No03: NOP   0;
NoXX: NOP   0;
NETWORK
TITLE =ASW_6030: Active step germinating
//      U     "MAL1S019Par".Par.FlagProcess.ProcessActive;
//      SPBN  tuen;
//
//// copy stepnr
//      L     "MAL1S019Par".Par.ParIntMachine.ActualStep;
//      T     "MAL1S019Par".Par.ParIntProcess.ActualStep;
//// set step conditions
//
//// Case where process is starting during loading
//      U     "MAL1S019Par".Par.FlagProcess.ProcessActive;
//      UN    "MAL1S019Par".Par.FlagFunction_1.StepLoading; // Step loading
//      SPBN  e003;
//// lifting devices must be in highest position
//      L       WinCoS_BIW01_09PLC1BIW01_02.Ma.Par.ParPositionTopRightUnits;
////Malting Plant OAO Belsolod Ivanonvo Weissrussland
//      L     50; // 50mm offset
//      +I    ;
//      T     "MAL1S019Par".Par.MachineValue.SOLLWERT_HUBZUG1_HOEHE;
//      L       WinCoS_BIW01_09PLC1BIW01_02.Ma.Par.ParPositionTopLeftUnits;
////Malting Plant OAO Belsolod Ivanonvo Weissrussland
//      L     50; // 50mm offset
//      +I    ;
//      T     "MAL1S019Par".Par.MachineValue.SOLLWERT_HUBZUG2_HOEHE;
//      L     5;
//      T     WinCoS_BIW01_09PLC1BIW01_02.Ma.Par.ParTolPosition;
//e003: NOP   0;
//
//// reset turning cmds
//
//// save turning cmds from prev.step
//      L     "MAL1S019Par".Par.ParIntMachine.ActualStep;
//      L     "MAL1S019Par".Par.ParIntProcess.PrevStep1stTurn;
//      <>I   ;
//      SPB   sav1;
//      U     "MAL1S019Par".Par.FlagProcess2.Turning1WithSpraying;
//      =     "MAL1S019Par".Par.Switches1.StaOn08; // Turning1WithSpraying
//      U     "MAL1S019Par".Par.FlagProcess2.Turning1WithDosing;
//      =     "MAL1S019Par".Par.Switches1.StaOn09; // Turning1WithDosing
//sav1: NOP   0;
//      L     "MAL1S019Par".Par.ParIntMachine.ActualStep;
//      L     "MAL1S019Par".Par.ParIntProcess.PrevStep2ndTurn;
//      <>I   ;
//      SPB   sav2;
//      U     "MAL1S019Par".Par.FlagProcess2.Turning2WithSpraying;
//      =     "MAL1S019Par".Par.Switches1.StaOn10; // Turning2WithSpraying
//      U     "MAL1S019Par".Par.FlagProcess2.Turning2WithDosing;
//      =     "MAL1S019Par".Par.Switches1.StaOn11; // Turning2WithDosing
//sav2: NOP   0;
//
//      SET   ;
//      R     "MAL1S019Par".Par.FlagProcess2.Turning1WithoutSpraying;
//      R     "MAL1S019Par".Par.FlagProcess2.Turning1WithSpraying;
//      R     "MAL1S019Par".Par.FlagProcess2.Turning1WithDosing;
//      R     "MAL1S019Par".Par.FlagProcess2.Turning2WithoutSpraying;
//      R     "MAL1S019Par".Par.FlagProcess2.Turning2WithSpraying;
//      R     "MAL1S019Par".Par.FlagProcess2.Turning2WithDosing;
//
//// Delta Temp to switch to next step
//      L     "MAL1S019Par".StepAct.DeltaTempSwitchpointStep;
//      L     L#0;
//      >D   ;
//      =     "MAL1S019Par".Par.FlagProcess1.DeltaTempNextStep;
//// Max Temp to switch to next step
//      L     "MAL1S019Par".StepAct.MaxTempAboveFloorStep;
//      L     L#0;
//      >D   ;
//      =     "MAL1S019Par".Par.FlagProcess1.MaxTempNextStep;
//
//// position waste air see sub 6050
//
//// basic speed fan see sub 6040
//
//// air humifidication
//      L     1;
//      L     "MAL1S019Par".StepAct.AirMoisten;   // On/Off
//      ==I;  // air humifidication on
//      U     WinCoS_BIW01_09PLC1BIW01_02.Ma.StStartedFwd; //Malting Plant OAO
//Belsolod Ivanonvo Weissrussland
//      =     "MAL1S019Par".Par.FlagProcess.AirHumidificationValve1; // air
//humifidication valve 1 on
//      U(    ; // air humifidication on
//      L     "MAL1S019Par".Par.ParIntMachine.TargetSpeedGermFan; // germinating
//fan is running
//      L     40; // fanspeed > 40%
//      >I    ; // muss noch in Istwert getauscht werden JV
//      )     ; // fanspeed > 40%
//      =     "MAL1S019Par".Par.FlagProcess.AirHumidificationValve2;
//
//// air cooling
//      L     "MAL1S019Par".StepAct.Cooling;
//      L   1;  // Activate Cooling System = 1 (yes)
//      ==I;
//      =     "MAL1S019Par".Par.FlagProcess.Cooling; // request cooling
//
//      U     "MAL1S019Par".Par.FlagProcess.ProcessActive;
//      U     "MAL1S019".PCRead.Step.StReady;
//      UN    "MAL1S019Par".Par.FlagFunction_1.StepLoading;
//      SPBN  e630;
//
//// turning 1
//      UN    "MAL1S019Par".Par.FlagProcess2.StartSecondTurningRound; // Turn
//from PrevStep
//      U(;
//      L     "MAL1S019Par".StepAct.StartTurningRound_1;
//      L     0;
//      >=D;                  // negative, no turning 1
//      );
//      U(    ;
//      O(    ; // Nach Rezept
//      L     "MAL1S019Par".ActTimeStepProcess.StepTimeActHourTotal; // Steptime
//in hours overall
//      L     "MAL1S019Par".StepAct.StartTurningRound_1;
//      ==I   ;
//      UN     WinCoS_BIW01_09PLC1BIW01_02.Ma.StAdjusted; // target position
//turning reached
//      )     ;
//      O(    ; // Selbsthaltung
//      L     "MAL1S019Par".ActTimeStepProcess.StepTimeActHourTotal; // Steptime
//in hours overall
//      L     "MAL1S019Par".StepAct.StartTurningRound_1;
//      <>I   ;
//      U     "MAL1S019Par".Par.FlagProcess2.StartFirstTurningRound;
//      )     ;
//      )     ;
//      S     "MAL1S019Par".Par.FlagProcess2.Turning1WithoutSpraying;
//      S     "MAL1S019Par".Par.FlagFunction_1.TurningStart;
//// turning 1 with spraying
//      U(    ;
//      L     1;
//      L     "MAL1S019Par".StepAct.TurningWithSpraying_1;
//      ==I;    // turning 1 with spraying on
//      U(    ;
//      L     "MAL1S019Par".Par.ParIntMachine.ActualStep;
//      L     "MAL1S019Par".Par.ParIntProcess.PrevStep1stTurn;
//      ==I   ;
//      )     ;
//      )     ;
//      O(    ;
//      L     "MAL1S019Par".Par.ParIntMachine.ActualStep;
//      L     "MAL1S019Par".Par.ParIntProcess.PrevStep1stTurn;
//      <>I   ;
//      U     "MAL1S019Par".Par.Switches1.StaOn08; // Turning1WithSpraying
//      )     ;
//      U     "MAL1S019Par".Par.FlagProcess2.Turning1WithoutSpraying;
//      S     "MAL1S019Par".Par.FlagProcess2.Turning1WithSpraying;
//// turning 1 with spraying and GA3
//      U(    ;
//      L     1;
//      L     "MAL1S019Par".StepAct.TurningWithDosing_1;
//      ==I;    // turning 1 with spraying on
//      U(    ;
//      L     "MAL1S019Par".Par.ParIntMachine.ActualStep;
//      L     "MAL1S019Par".Par.ParIntProcess.PrevStep1stTurn;
//      ==I   ;
//      )     ;
//      )     ;
//      O(    ;
//      L     "MAL1S019Par".Par.ParIntMachine.ActualStep;
//      L     "MAL1S019Par".Par.ParIntProcess.PrevStep1stTurn;
//      <>I   ;
//      U     "MAL1S019Par".Par.Switches1.StaOn09; // Turning1WithDosing
//      )     ;
//      U     "MAL1S019Par".Par.FlagProcess2.Turning1WithoutSpraying;
//      S     "MAL1S019Par".Par.FlagProcess2.Turning1WithSpraying;
//      S     "MAL1S019Par".Par.FlagProcess2.Turning1WithDosing;
//
//      U     "MAL1S019Par".Par.FlagProcess2.Turning1WithoutSpraying;
//      U     "MAL1S019Par".Par.FlagFunction_1.TurningStart;
//      UN     WinCoS_BIW01_09PLC1BIW01_02.Ma.StAdjusted; // target position
//turning reached
//      FP    "MAL1S019Par".Par.FlagProcess2.StartFirstTurningFP;
//      S     "MAL1S019Par".Par.FlagProcess2.StartFirstTurningRound;
//
//      U     WinCoS_BIW01_09PLC1BIW01_02.Ma.StAdjusted; // target position
//turning reached
//      O(    ;
//      L     "MAL1S019Par".ActTimeStepProcess.StepTimeActHourTotal; // Steptime
//in hours overall
//      L     "MAL1S019Par".StepAct.StartTurningRound_1;
//      >I    ;
//      U     WinCoS_BIW01_09PLC1BIW01_02.Ma.StAdjusted; // target position
//turning reached
//      )     ;
//      U     "MAL1S019Par".Par.FlagProcess2.StartFirstTurningRound;
//      R     "MAL1S019Par".Par.FlagProcess2.StartFirstTurningRound;
//
//      U     "MAL1S019Par".Par.FlagProcess2.StartFirstTurningFP;
//      SPB   trn1;
//      L     "MAL1S019Par".Par.ParIntMachine.ActualStep;
//      T     "MAL1S019Par".Par.ParIntProcess.PrevStep1stTurn;
//trn1: NOP   0;
//
//// turning 2
//      UN    "MAL1S019Par".Par.FlagProcess2.StartFirstTurningRound; // Unsinngie
//Rezeptwerte
//      U(;
//      L     1;
//      L     "MAL1S019Par".StepAct.StartTurningRound_2;
//      ==I    ;
//      );
//      U(    ;
//      O(    ; // Nach Rezept
//      L     "MAL1S019Par".ActTimeStepProcess.StepTimeActHourTotal; // Steptime
//in hours overall
//      L     "MAL1S019Par".StepAct.StartTurningRound_2;
//      ==I   ;
//      UN     WinCoS_BIW01_09PLC1BIW01_02.Ma.StAdjusted; // target position
//turning reached
//      )     ;
//      O(    ; // Selbsthaltung
//      L     "MAL1S019Par".ActTimeStepProcess.StepTimeActHourTotal; // Steptime
//in hours overall
//      L     "MAL1S019Par".StepAct.StartTurningRound_2;
//      <>I   ;
//      U     "MAL1S019Par".Par.FlagProcess2.StartSecondTurningRound;
//      )     ;
//      )     ;
//      S     "MAL1S019Par".Par.FlagProcess2.Turning2WithoutSpraying;
//      S     "MAL1S019Par".Par.FlagFunction_1.TurningStart;
//// turning 2 with spraying
//      U(    ;
//      L     1;
//      L     "MAL1S019Par".StepAct.TurningWithSpraying_2;
//      ==I    ;
//      U(    ;
//      L     "MAL1S019Par".Par.ParIntMachine.ActualStep;
//      L     "MAL1S019Par".Par.ParIntProcess.PrevStep2ndTurn;
//      ==I   ;
//      )     ;
//      )     ;
//      O(    ;
//      L     "MAL1S019Par".Par.ParIntMachine.ActualStep;
//      L     "MAL1S019Par".Par.ParIntProcess.PrevStep2ndTurn;
//      <>I   ;
//      U     "MAL1S019Par".Par.Switches1.StaOn10; // Turning2WithSpraying
//      )     ;
//      U     "MAL1S019Par".Par.FlagProcess2.Turning2WithoutSpraying;
//      S     "MAL1S019Par".Par.FlagProcess2.Turning2WithSpraying;
//// turning 2 with spraying and GA3
//      U(    ;
//      L     1;
//      L     "MAL1S019Par".StepAct.TurningWithDosing_2;
//      ==I;    // turning 2 with spraying and GA3 on
//      U(    ;
//      L     "MAL1S019Par".Par.ParIntMachine.ActualStep;
//      L     "MAL1S019Par".Par.ParIntProcess.PrevStep2ndTurn;
//      ==I   ;
//      )     ;
//      )     ;
//      O(    ;
//      L     "MAL1S019Par".Par.ParIntMachine.ActualStep;
//      L     "MAL1S019Par".Par.ParIntProcess.PrevStep2ndTurn;
//      <>I   ;
//      U     "MAL1S019Par".Par.Switches1.StaOn11; // Turning2WithDosing
//      )     ;
//      U     "MAL1S019Par".Par.FlagProcess2.Turning2WithoutSpraying;
//      S     "MAL1S019Par".Par.FlagProcess2.Turning2WithSpraying;
//      S     "MAL1S019Par".Par.FlagProcess2.Turning2WithDosing;
//
//      U     "MAL1S019Par".Par.FlagProcess2.Turning2WithoutSpraying;
//      U     "MAL1S019Par".Par.FlagFunction_1.TurningStart;
//      UN     WinCoS_BIW01_09PLC1BIW01_02.Ma.StAdjusted; // target position
//turning reached
//      FP    "MAL1S019Par".Par.FlagProcess2.StartSecondTurningFP;
//      S     "MAL1S019Par".Par.FlagProcess2.StartSecondTurningRound;
//
//      U     WinCoS_BIW01_09PLC1BIW01_02.Ma.StAdjusted; // target position
//turning reached
//      O(    ;
//      L     "MAL1S019Par".ActTimeStepProcess.StepTimeActHourTotal; // Steptime
//in hours overall
//      L     "MAL1S019Par".StepAct.StartTurningRound_2;
//      >I    ;
//      U     WinCoS_BIW01_09PLC1BIW01_02.Ma.StAdjusted; // target position
//turning reached
//      )     ;
//      U     "MAL1S019Par".Par.FlagProcess2.StartSecondTurningRound;
//      R     "MAL1S019Par".Par.FlagProcess2.StartSecondTurningRound;
//
//      U     "MAL1S019Par".Par.FlagProcess2.StartSecondTurningFP;
//      SPB   trn2;
//      L     "MAL1S019Par".Par.ParIntMachine.ActualStep;
//      T     "MAL1S019Par".Par.ParIntProcess.PrevStep2ndTurn;
//trn2: NOP   0;
////Fix Speed for Turning
//      U     "MAL1S019Par".Par.FlagProcess2.Turning1WithoutSpraying;
//      O     "MAL1S019Par".Par.FlagProcess2.Turning1WithSpraying;
//      O     "MAL1S019Par".Par.FlagProcess2.Turning2WithoutSpraying;
//      O     "MAL1S019Par".Par.FlagProcess2.Turning2WithSpraying;
//      U    M 50.0;
//      SPBN  SpdT;
//      L     15; // 15Hz
//      T     "MAL1S019Par".Par.MachineValue.SollwertFahrantrieb;
//SpdT: NOP   0;
//
//// find turning direction
//      U     "MAL1S019Par".Par.FlagGen.TurningStarted;
//      O(    ;
//      UN    "MAL1S019Par".Par.FlagProcess2.Turning1WithoutSpraying;
//      UN    "MAL1S019Par".Par.FlagProcess2.Turning2WithoutSpraying;
//      )     ;
//      SPB   tuen;
//      L     "MAL1S019Par".Par.ParIntMachine.TargetPosTravDriTurnRigt; // 370° =
//endposition turning right
//      T     WinCoS_BIW01_09PLC1BIW01_02.Ma.InPositionTarget; // target position
//turning reached
//
//      U(    ;
//      L     WinCoS_BIW01_09PLC1BIW01_02.Ma.OutPositionAngle;
//      L     1800;
//      <I    ; // condition turning right (clockwise)
//      )     ;
//      S     "MAL1S019Par".Par.FlagFunction_1.TurningRight;
//      S     "MAL1S019Par".Par.FlagGen.TurningStarted;
//// - Correct effect of ILO Mode
//      L       WinCoS_BIW01_09PLC1BIW01_02.Ma.Par.ParPositionTopLeftUnits;
////Malting Plant OAO Belsolod Ivanonvo Weissrussland
//      T     "MAL1S019Par".Par.MachineValue.SOLLWERT_HUBZUG1_HOEHE;
//      L       WinCoS_BIW01_09PLC1BIW01_02.Ma.Par.ParPositionTopRightUnits;
////Malting Plant OAO Belsolod Ivanonvo Weissrussland
//      T     "MAL1S019Par".Par.MachineValue.SOLLWERT_HUBZUG2_HOEHE;
//      SPB   E603   ;
//      L     "MAL1S019Par".Par.ParIntMachine.TargetPosTravDriTurnLeft; // 0° =
//endposition turning left
//      T     WinCoS_BIW01_09PLC1BIW01_02.Ma.InPositionTarget; // target position
//turning reached
//
//      U(    ;
//      L     WinCoS_BIW01_09PLC1BIW01_02.Ma.OutPositionAngle;
//      L     1800;
//      >=I   ; // condition turning left (counterclockwise)
//      )     ;
//      S     "MAL1S019Par".Par.FlagFunction_1.TurningLeft;
//      S     "MAL1S019Par".Par.FlagGen.TurningStarted;
//// - Correct effect of ILO Mode
//      L       WinCoS_BIW01_09PLC1BIW01_02.Ma.Par.ParPositionTopLeftUnits;
////Malting Plant OAO Belsolod Ivanonvo Weissrussland
//      T     "MAL1S019Par".Par.MachineValue.SOLLWERT_HUBZUG1_HOEHE;
//      L       WinCoS_BIW01_09PLC1BIW01_02.Ma.Par.ParPositionTopRightUnits;
////Malting Plant OAO Belsolod Ivanonvo Weissrussland
//      T     "MAL1S019Par".Par.MachineValue.SOLLWERT_HUBZUG2_HOEHE;
//      SPB   E603   ;
//tuen: NOP   0;
//// - Case of fast speed to protect a 2nd start during same hours as finsihed
//      O(    ; // Nach Rezept
//      L     "MAL1S019Par".ActTimeStepProcess.StepTimeActHourTotal; // Steptime
//in hours overall
//      L     "MAL1S019Par".StepAct.StartTurningRound_1;
//      ==I   ;
//      U     WinCoS_BIW01_09PLC1BIW01_02.Ma.StAdjusted; // target position
//turning reached
//      U     "MAL1S019Par".Par.FlagFunction_1.TurningStart;
//      )     ;
//      O(    ; // Nach Rezept
//      L     "MAL1S019Par".ActTimeStepProcess.StepTimeActHourTotal; // Steptime
//in hours overall
//      L     "MAL1S019Par".StepAct.StartTurningRound_2;
//      ==I   ;
//      U     WinCoS_BIW01_09PLC1BIW01_02.Ma.StAdjusted; // target position
//turning reached
//      U     "MAL1S019Par".Par.FlagFunction_1.TurningStart;
//      )     ;
//      SPB   e603;
//
//// reset turning right (clockwise)
//      U     "MAL1S019Par".Par.FlagFunction_1.TurningRight;
//      U(    ;
//      O      WinCoS_BIW01_09PLC1BIW01_02.Ma.StAdjusted; // target position
//turning reached
//      O(    ;
//      L     WinCoS_BIW01_09PLC1BIW01_02.Ma.OutPositionAngle;
//      L     WinCoS_BIW01_09PLC1BIW01_02.Ma.Par.ParTolPosition;
//      +I    ;
//      L     "MAL1S019Par".Par.ParIntMachine.TargetPosTravDriTurnRigt;
//      >=I   ;
//      )     ;
//      )     ;
//      R     "MAL1S019Par".Par.FlagFunction_1.TurningRight;
//      R     "MAL1S019Par".Par.FlagFunction_1.TurningStart;
//
//// reset turning left (counterclockwise)
//      U     "MAL1S019Par".Par.FlagFunction_1.TurningLeft;
//      U(    ;
//      O     WinCoS_BIW01_09PLC1BIW01_02.Ma.StAdjusted; // target position
//turning reached
//      O(    ;
//      L     WinCoS_BIW01_09PLC1BIW01_02.Ma.OutPositionAngle;
//      L     WinCoS_BIW01_09PLC1BIW01_02.Ma.Par.ParTolPosition;
//      -I    ;
//      L     "MAL1S019Par".Par.ParIntMachine.TargetPosTravDriTurnLeft;
//      <=I   ;
//      )     ;
//      )     ;
//      R     "MAL1S019Par".Par.FlagFunction_1.TurningLeft;
//      R     "MAL1S019Par".Par.FlagFunction_1.TurningStart;
//
//// reset turning flag
//      U     "MAL1S019Par".Par.FlagGen.TurningStarted;
//      UN    "MAL1S019Par".Par.FlagProcess2.Turning1WithoutSpraying;
//      UN    "MAL1S019Par".Par.FlagProcess2.Turning2WithoutSpraying;
//      O(    ;
//      U     "MAL1S019Par".Par.FlagGen.TurningStarted;
//      U     WinCoS_BIW01_09PLC1BIW01_02.Ma.StAdjusted; // target position
//turning reached
//      )     ;
//      ON    "MAL1S019Par".Par.FlagProcess.ProcessActive;
//      R     "MAL1S019Par".Par.FlagGen.TurningStarted;
//      R     "MAL1S019Par".Par.FlagProcess2.Turning1WithoutSpraying;
//      R     "MAL1S019Par".Par.FlagProcess2.Turning2WithoutSpraying;
//      R     "MAL1S019Par".Par.FlagFunction_1.TurningStart;
//e630: NOP   0;
//      UN    "MAL1S019Par".Par.FlagProcess.ProcessActive;
//      R     "MAL1S019Par".Par.FlagProcess2.StartFirstTurningRound;
//      R     "MAL1S019Par".Par.FlagProcess2.StartSecondTurningRound;
//
//e603: NOP   0;
//E603: NOP   0;

      A     "MAL1S019Par".Par.FlagProcess.ProcessActive;
      JCN   tuen;

// copy stepnr
      L     "MAL1S019Par".Par.ParIntMachine.ActualStep;
      T     "MAL1S019Par".Par.ParIntProcess.ActualStep;
// set step conditions

// reset turning cmds

// save turning cmds from prev.step
      L     "MAL1S019Par".Par.ParIntMachine.ActualStep;
      L     "MAL1S019Par".Par.ParIntProcess.PrevStep1stTurn;
      <>I   ;
      JC    sav1;
      A     "MAL1S019Par".Par.FlagProcess2.Turning1WithSpraying;
      =     "MAL1S019Par".Par.Switches1.StaOn08; // Turning1WithSpraying
      A     "MAL1S019Par".Par.FlagProcess2.Turning1WithDosing;
      =     "MAL1S019Par".Par.Switches1.StaOn09; // Turning1WithDosing
sav1: NOP   0;
      L     "MAL1S019Par".Par.ParIntMachine.ActualStep;
      L     "MAL1S019Par".Par.ParIntProcess.PrevStep2ndTurn;
      <>I   ;
      JC    sav2;
      A     "MAL1S019Par".Par.FlagProcess2.Turning2WithSpraying;
      =     "MAL1S019Par".Par.Switches1.StaOn10; // Turning2WithSpraying
      A     "MAL1S019Par".Par.FlagProcess2.Turning2WithDosing;
      =     "MAL1S019Par".Par.Switches1.StaOn11; // Turning2WithDosing
sav2: NOP   0;

      SET   ;
      R     "MAL1S019Par".Par.FlagProcess2.Turning1WithoutSpraying;
      R     "MAL1S019Par".Par.FlagProcess2.Turning1WithSpraying;
      R     "MAL1S019Par".Par.FlagProcess2.Turning1WithDosing;
      R     "MAL1S019Par".Par.FlagProcess2.Turning2WithoutSpraying;
      R     "MAL1S019Par".Par.FlagProcess2.Turning2WithSpraying;
      R     "MAL1S019Par".Par.FlagProcess2.Turning2WithDosing;

// Delta Temp to switch to next step
      L     "MAL1S019Par".StepAct.DeltaTempSwitchpointStep;
      L     L#0;
      >D    ;
      =     "MAL1S019Par".Par.FlagProcess1.DeltaTempNextStep;
// Max Temp to switch to next step
      L     "MAL1S019Par".StepAct.MaxTempAboveFloorStep;
      L     L#0;
      >D    ;
      =     "MAL1S019Par".Par.FlagProcess1.MaxTempNextStep;

// position waste air see sub 6050

// basic speed fan see sub 6040

// air humifidication

// air cooling
      L     "MAL1S019Par".StepAct.Cooling;
      L     1; // Activate Cooling System = 1 (yes)
      ==I   ;
      =     "MAL1S019Par".Par.FlagProcess.Cooling; // request cooling

      A     "MAL1S019Par".Par.FlagProcess.ProcessActive;
      A     "MAL1S019".PCRead.Step.StReady;
      AN    "MAL1S019Par".Par.FlagFunction_1.StepLoading;
      JCN   e630;

// turning 1
      AN    "MAL1S019Par".Par.FlagProcess2.StartSecondTurningRound; // Turn from PrevStep
      A(    ;
      L     "MAL1S019Par".StepAct.StartTurningRound_1;
      L     0;
      >=I   ; // negative, no turning 1
      )     ;
      A(    ;
      O(    ; // Nach Rezept
      L     "MAL1S019Par".ActTimeStepProcess.StepTimeActHourTotal; // Steptime in hours overall
      L     "MAL1S019Par".StepAct.StartTurningRound_1;
      ==I   ;
      AN    "G145M".A_2311_MXZ41MA.Ma.StAdjusted; // target position turning reached
      )     ;
      O(    ; // Selbsthaltung
      L     "MAL1S019Par".ActTimeStepProcess.StepTimeActHourTotal; // Steptime in hours overall
      L     "MAL1S019Par".StepAct.StartTurningRound_1;
      <>I   ;
      A     "MAL1S019Par".Par.FlagProcess2.StartFirstTurningRound;
      )     ;
      )     ;
      S     "MAL1S019Par".Par.FlagProcess2.Turning1WithoutSpraying;
      S     "MAL1S019Par".Par.FlagFunction_1.TurningStart;
// turning 1 with spraying
      A(    ;
      L     1;
      L     "MAL1S019Par".StepAct.TurningWithSpraying_1;
      ==I   ; // turning 1 with spraying on
      A(    ;
      L     "MAL1S019Par".Par.ParIntMachine.ActualStep;
      L     "MAL1S019Par".Par.ParIntProcess.PrevStep1stTurn;
      ==I   ;
      )     ;
      )     ;
      O(    ;
      L     "MAL1S019Par".Par.ParIntMachine.ActualStep;
      L     "MAL1S019Par".Par.ParIntProcess.PrevStep1stTurn;
      <>I   ;
      A     "MAL1S019Par".Par.Switches1.StaOn08; // Turning1WithSpraying
      )     ;
      A     "MAL1S019Par".Par.FlagProcess2.Turning1WithoutSpraying;
      S     "MAL1S019Par".Par.FlagProcess2.Turning1WithSpraying;
// turning 1 with spraying and GA3
      A(    ;
      L     1;
      L     "MAL1S019Par".StepAct.TurningWithDosing_1;
      ==I   ; // turning 1 with spraying on
      A(    ;
      L     "MAL1S019Par".Par.ParIntMachine.ActualStep;
      L     "MAL1S019Par".Par.ParIntProcess.PrevStep1stTurn;
      ==I   ;
      )     ;
      )     ;
      O(    ;
      L     "MAL1S019Par".Par.ParIntMachine.ActualStep;
      L     "MAL1S019Par".Par.ParIntProcess.PrevStep1stTurn;
      <>I   ;
      A     "MAL1S019Par".Par.Switches1.StaOn09; // Turning1WithDosing
      )     ;
      A     "MAL1S019Par".Par.FlagProcess2.Turning1WithoutSpraying;
      S     "MAL1S019Par".Par.FlagProcess2.Turning1WithSpraying;
      S     "MAL1S019Par".Par.FlagProcess2.Turning1WithDosing;

//BRT070410 - wird einen Zyklus später gesetzt
      A     "MAL1S019Par".Par.FlagProcess2.StartFirstDosingFP;
      S     "MAL1S019Par".Par.FlagProcess2.StartFirstTurningRound;

      A     "MAL1S019Par".Par.FlagProcess2.Turning1WithoutSpraying;
      A     "MAL1S019Par".Par.FlagFunction_1.TurningStart;
//BRT060310      UN    "G145M".A_2311_MXZ41MA.Ma.StAdjusted    // target position turning reached
      AN    "G145M".A_2311_MXZ41MA.Ma.OutAdjusted; // target position turning reached
      FP    "MAL1S019Par".Par.FlagProcess2.StartFirstTurningFP;
      =     "MAL1S019Par".Par.FlagProcess2.StartFirstDosingFP;
//BRT070410      S     "MAL1S019Par".Par.FlagProcess2.StartFirstTurningRound

      A     "MAL1S019Par".Par.FlagProcess2.StartFirstDosingFP;
      A     "MAL1S019Par".Par.FlagProcess2.StartFirstTurningFP;
      JCN   trn1;
      L     "MAL1S019Par".Par.ParIntMachine.ActualStep;
      T     "MAL1S019Par".Par.ParIntProcess.PrevStep1stTurn;
trn1: NOP   0;

//BRT060310      U    "G145M".A_2311_MXZ41MA.Ma.StAdjusted    // target position turning reached
      A     "G145M".A_2311_MXZ41MA.Ma.OutAdjusted; // target position turning reached
      O(    ;
      L     "MAL1S019Par".ActTimeStepProcess.StepTimeActHourTotal; // Steptime in hours overall
      L     "MAL1S019Par".StepAct.StartTurningRound_1;
      >I    ;
      A(    ;
      O     "G145M".A_2311_MXZ41MA.Ma.OutAdjusted; // target position turning reached
      O(    ;
//BRT070310      UN    "G145M".A_2311_BZS46.StTrue // stop fan side
//BRT070310      U     "G145M".A_2311_BZS44.StTrue // stop discharge side
      A     "G145M".A_2311_BZS46.StTrue; // stop end side
      AN    "G145M".A_2311_BZS44.StTrue; // stop zeroposition
      A     "MAL1S019Par".Par.FlagFunction_1.TurningRight;
      )     ;
      O(    ;
//BRT070310      U     "G145M".A_2311_BZS46.StTrue // stop fan side
//BRT070310      UN    "G145M".A_2311_BZS44.StTrue // stop discharge side
      AN    "G145M".A_2311_BZS46.StTrue; // stop end side
      A     "G145M".A_2311_BZS44.StTrue; // stop zeroposition
      A     "MAL1S019Par".Par.FlagFunction_1.TurningLeft;
      )     ;
      )     ;
      )     ;
      O(    ;
      L     "MAL1S019Par".StepAct.StartTurningRound_1;
//BRT070310      L     0
//BRT070310      <D                                // negative, no turning 1
      L     -1; //BRT070310
      ==I   ; //BRT070310
      )     ;
      A     "MAL1S019Par".Par.FlagProcess2.StartFirstTurningRound;
      R     "MAL1S019Par".Par.FlagProcess2.StartFirstTurningRound;
      R     "MAL1S019Par".Par.Switches1.StaOn08; // Turning1WithSpraying
      R     "MAL1S019Par".Par.Switches1.StaOn09; // Turning1WithDosing

// turning 2
      AN    "MAL1S019Par".Par.FlagProcess2.StartFirstTurningRound; // Unsinnige Rezeptwerte
      A(    ;
      L     "MAL1S019Par".StepAct.StartTurningRound_2;
      L     0;
      >=I   ;
      )     ;
      A(    ;
      O(    ; // Nach Rezept
      L     "MAL1S019Par".ActTimeStepProcess.StepTimeActHourTotal; // Steptime in hours overall
      L     "MAL1S019Par".StepAct.StartTurningRound_2;
      ==I   ;
      AN    "G145M".A_2311_MXZ41MA.Ma.StAdjusted; // target position turning reached
      )     ;
      O(    ; // Selbsthaltung
      L     "MAL1S019Par".ActTimeStepProcess.StepTimeActHourTotal; // Steptime in hours overall
      L     "MAL1S019Par".StepAct.StartTurningRound_2;
      <>I   ;
      A     "MAL1S019Par".Par.FlagProcess2.StartSecondTurningRound;
      )     ;
      )     ;
      S     "MAL1S019Par".Par.FlagProcess2.Turning2WithoutSpraying;
      S     "MAL1S019Par".Par.FlagFunction_1.TurningStart;
// turning 2 with spraying
      A(    ;
      L     1;
      L     "MAL1S019Par".StepAct.TurningWithSpraying_2;
      ==I   ;
      A(    ;
      L     "MAL1S019Par".Par.ParIntMachine.ActualStep;
      L     "MAL1S019Par".Par.ParIntProcess.PrevStep2ndTurn;
      ==I   ;
      )     ;
      )     ;
      O(    ;
      L     "MAL1S019Par".Par.ParIntMachine.ActualStep;
      L     "MAL1S019Par".Par.ParIntProcess.PrevStep2ndTurn;
      <>I   ;
      A     "MAL1S019Par".Par.Switches1.StaOn10; // Turning2WithSpraying
      )     ;
      A     "MAL1S019Par".Par.FlagProcess2.Turning2WithoutSpraying;
      S     "MAL1S019Par".Par.FlagProcess2.Turning2WithSpraying;
// turning 2 with spraying and GA3
      A(    ;
      L     1;
      L     "MAL1S019Par".StepAct.TurningWithDosing_2;
      ==I   ; // turning 2 with spraying and GA3 on
      A(    ;
      L     "MAL1S019Par".Par.ParIntMachine.ActualStep;
      L     "MAL1S019Par".Par.ParIntProcess.PrevStep2ndTurn;
      ==I   ;
      )     ;
      )     ;
      O(    ;
      L     "MAL1S019Par".Par.ParIntMachine.ActualStep;
      L     "MAL1S019Par".Par.ParIntProcess.PrevStep2ndTurn;
      <>I   ;
      A     "MAL1S019Par".Par.Switches1.StaOn11; // Turning2WithDosing
      )     ;
      A     "MAL1S019Par".Par.FlagProcess2.Turning2WithoutSpraying;
      S     "MAL1S019Par".Par.FlagProcess2.Turning2WithSpraying;
      S     "MAL1S019Par".Par.FlagProcess2.Turning2WithDosing;

//BRT070410 - wird einen Zyklus später gesetzt
      A     "MAL1S019Par".Par.FlagProcess2.StartSecondDosingFP;
      S     "MAL1S019Par".Par.FlagProcess2.StartSecondTurningRound;

      A     "MAL1S019Par".Par.FlagProcess2.Turning2WithoutSpraying;
      A     "MAL1S019Par".Par.FlagFunction_1.TurningStart;
//BRT060310      UN    "G145M".A_2311_MXZ41MA.Ma.StAdjusted    // target position turning reached
      AN    "G145M".A_2311_MXZ41MA.Ma.OutAdjusted; // target position turning reached
      FP    "MAL1S019Par".Par.FlagProcess2.StartSecondTurningFP;
      =     "MAL1S019Par".Par.FlagProcess2.StartSecondDosingFP;
//BRT070410      S     "MAL1S019Par".Par.FlagProcess2.StartSecondTurningRound

      A     "MAL1S019Par".Par.FlagProcess2.StartSecondDosingFP;
      A     "MAL1S019Par".Par.FlagProcess2.StartSecondTurningFP;
      JCN   trn2;
      L     "MAL1S019Par".Par.ParIntMachine.ActualStep;
      T     "MAL1S019Par".Par.ParIntProcess.PrevStep2ndTurn;
trn2: NOP   0;

//BRT060310      U    "G145M".A_2311_MXZ41MA.Ma.StAdjusted    // target position turning reached
      A     "G145M".A_2311_MXZ41MA.Ma.OutAdjusted; // target position turning reached
      O(    ;
      L     "MAL1S019Par".ActTimeStepProcess.StepTimeActHourTotal; // Steptime in hours overall
      L     "MAL1S019Par".StepAct.StartTurningRound_2;
      >I    ;
      A(    ;
      O     "G145M".A_2311_MXZ41MA.Ma.OutAdjusted; // target position turning reached
      O(    ;
      AN    "G145M".A_2311_BZS46.StTrue; // stop fan side
      A     "G145M".A_2311_BZS44.StTrue; // stop discharge side
      A     "MAL1S019Par".Par.FlagFunction_1.TurningRight;
      )     ;
      O(    ;
      A     "G145M".A_2311_BZS46.StTrue; // stop fan side
      AN    "G145M".A_2311_BZS44.StTrue; // stop discharge side
      A     "MAL1S019Par".Par.FlagFunction_1.TurningLeft;
      )     ;
      )     ;
      )     ;
      O(    ;
      L     "MAL1S019Par".StepAct.StartTurningRound_2;
//BRT070310      L     0
//BRT070310      <D                                // negative, no turning 2
      L     -1; //BRT070310
      ==I   ; //BRT070310
      )     ;
      A     "MAL1S019Par".Par.FlagProcess2.StartSecondTurningRound;
      R     "MAL1S019Par".Par.FlagProcess2.StartSecondTurningRound;
      R     "MAL1S019Par".Par.Switches1.StaOn10; // Turning2WithSpraying
      R     "MAL1S019Par".Par.Switches1.StaOn11; // Turning2WithDosing

      L     3600;
      T     "MAL1S019Par".Par.ParIntMachine.TargetPosTravDriTurnRigt; // 360° = endposition turning right

// find turning direction spez. APU: right ==> forward, left ==> reverse
      A     "MAL1S019Par".Par.FlagGen.TurningStarted;
      O(    ;
      AN    "MAL1S019Par".Par.FlagProcess2.Turning1WithoutSpraying;
      AN    "MAL1S019Par".Par.FlagProcess2.Turning2WithoutSpraying;
      )     ;
      JC    tuen;
      L     "MAL1S019Par".Par.ParIntMachine.TargetPosTravDriTurnRigt; // 360° = endposition turning right
      T     "G145M".A_2311_MXZ41MA.Ma.InPositionTarget; // target position turning

      A(    ;
      L     "G145M".A_2311_MXZ41MA.Ma.OutPositionAngle;
      L     1800;
      <I    ; // condition turning right (clockwise)
      )     ;
//BRT070310      O     "G145M".A_2311_BZS46.StTrue // stop end side
//BRT070310      UN    "G145M".A_2311_BZS44.StTrue // stop zeroposition
      O     "G145M".A_2311_BZS44.StTrue; // stop zeroposition  //BRT070310
      AN    "G145M".A_2311_BZS46.StTrue; //stop end side   //BRT070310
      S     "MAL1S019Par".Par.FlagFunction_1.TurningRight;
      S     "MAL1S019Par".Par.FlagGen.TurningStarted;
      JC    E603;
      L     "MAL1S019Par".Par.ParIntMachine.TargetPosTravDriTurnLeft; // 0° = endposition turning left
      T     "G145M".A_2311_MXZ41MA.Ma.InPositionTarget; // target position turning

      A(    ;
      L     "G145M".A_2311_MXZ41MA.Ma.OutPositionAngle;
      L     1800;
      >=I   ; // condition turning left (counterclockwise)
      )     ;
//BRT070310      O     "G145M".A_2311_BZS44.StTrue // stop end side
//BRT070310      UN    "G145M".A_2311_BZS46.StTrue // stop zeroposition
      O     "G145M".A_2311_BZS46.StTrue; // stop zeroposition  //BRT070310
      AN    "G145M".A_2311_BZS44.StTrue; //stop end side   //BRT070310
      S     "MAL1S019Par".Par.FlagFunction_1.TurningLeft;
      S     "MAL1S019Par".Par.FlagGen.TurningStarted;
      JC    E603;
tuen: NOP   0;

// reset turning right (clockwise)
      A     "MAL1S019Par".Par.FlagFunction_1.TurningRight;
      A(    ;
//      O     "G202M"._2111_MXZ41MA.Ma.StAdjusted    // target position turning reached
      O(    ;
      L     "G145M".A_2311_MXZ41MA.Ma.OutPositionAngle;
      L     "G145M".A_2311_MXZ41MA.Ma.Par.ParTolPosition;
      +I    ;
      L     "MAL1S019Par".Par.ParIntMachine.TargetPosTravDriTurnRigt;
      >=I   ;
      )     ;
//BRT070310      O     "G145M".A_2311_BZS44.StTrue // stop end side
      O     "G145M".A_2311_BZS46.StTrue; // stop zeroposition
      )     ;
      R     "MAL1S019Par".Par.FlagFunction_1.TurningRight;
      R     "MAL1S019Par".Par.FlagFunction_1.TurningStart;

// reset turning left (counterclockwise)
      A     "MAL1S019Par".Par.FlagFunction_1.TurningLeft;
      A(    ;
//      O     "G202M"._2111_MXZ41MA.Ma.StAdjusted    // target position turning reached
      O(    ;
      L     "G145M".A_2311_MXZ41MA.Ma.OutPositionAngle;
      L     "G145M".A_2311_MXZ41MA.Ma.Par.ParTolPosition;
      -I    ;
      L     "MAL1S019Par".Par.ParIntMachine.TargetPosTravDriTurnLeft;
      <=I   ;
      )     ;
      O     "G145M".A_2311_BZS44.StTrue; // stop end side
//BRT070310      O     "G145M".A_2311_BZS46.StTrue // stop zeroposition
      )     ;
      R     "MAL1S019Par".Par.FlagFunction_1.TurningLeft;
      R     "MAL1S019Par".Par.FlagFunction_1.TurningStart;

// - Case of fast speed to protect a 2nd start during same hours as finsihed
      A     "MAL1S019Par".Par.FlagGen.TurningStarted;
//====>BRT070310      UN    "MAL1S019Par".Par.FlagProcess.ProcessEnd    // JV210808 to finish last turning
      A(    ;
      A     "MAL1S019Par".Par.FlagProcess2.Turning1WithoutSpraying;
      O     "MAL1S019Par".Par.FlagProcess2.Turning2WithoutSpraying;
      AN    "MAL1S019Par".Par.FlagProcess.ProcessEnd; // JV210808 to finish last turning
      )     ;
      AN    "MAL1S019StepValues".StartStep; // start step for average calculating
      A(    ;
      O(    ; // Nach Rezept
      A(    ;
      L     "MAL1S019Par".ActTimeStepProcess.StepTimeActHourTotal; // Steptime in hours overall
      L     "MAL1S019Par".StepAct.StartTurningRound_1;
      ==I   ; // JV 250808
      )     ;
//      UN    "MAL1S019Par".Par.FlagProcess2.StartFirstTurningRound    // JV 250808
      A     "G145M".A_2311_MXZ41MA.Ma.OutAdjusted; // target position turning reached
      )     ;
      O(    ; // Nach Rezept
      A(    ;
      L     "MAL1S019Par".ActTimeStepProcess.StepTimeActHourTotal; // Steptime in hours overall
      L     "MAL1S019Par".StepAct.StartTurningRound_2;
      ==I   ; // JV 250808
      )     ;
//      UN    "MAL1S019Par".Par.FlagProcess2.StartSecondTurningRound    // JV 250808
      A     "G145M".A_2311_MXZ41MA.Ma.OutAdjusted; // target position turning reached
//<====BRT070310
      )     ;
      )     ;
      O(    ;
      AN    "G145M".A_2311_MXZ41MA.Ma.OutAdjusted; // target position turning reached
      AN    "MAL1S019Par".Par.FlagFunction_1.StepUnloading;
      )     ;
      JC    e603;

// reset turning flag
      A     "MAL1S019Par".Par.FlagGen.TurningStarted;
      ON    "MAL1S019Par".Par.FlagProcess.ProcessActive;
      R     "MAL1S019Par".Par.FlagGen.TurningStarted;
      R     "MAL1S019Par".Par.FlagProcess2.Turning1WithoutSpraying;
      R     "MAL1S019Par".Par.FlagProcess2.Turning2WithoutSpraying;
      R     "MAL1S019Par".Par.FlagProcess2.Turning1WithSpraying;
      R     "MAL1S019Par".Par.FlagProcess2.Turning2WithSpraying;
      R     "MAL1S019Par".Par.FlagProcess2.Turning1WithDosing;
      R     "MAL1S019Par".Par.FlagProcess2.Turning2WithDosing;
      R     "MAL1S019Par".Par.FlagFunction_1.TurningStart;
      R     "MAL1S019Par".Par.FlagProcess2.StartFirstTurningRound; // JV 250808
      R     "MAL1S019Par".Par.FlagProcess2.StartSecondTurningRound; // JV 250808
      SET   ;
      R     "MAL1S019StepValues".StartStep; // start step for average calculating
e630: NOP   0;
      AN    "MAL1S019Par".Par.FlagProcess.ProcessActive;
      R     "MAL1S019Par".Par.FlagProcess2.StartFirstTurningRound;
      R     "MAL1S019Par".Par.FlagProcess2.StartSecondTurningRound;
      R     "MAL1S019Par".Par.Switches1.StaOn08; // Turning1WithSpraying
      R     "MAL1S019Par".Par.Switches1.StaOn09; // Turning1WithDosing
      R     "MAL1S019Par".Par.Switches1.StaOn10; // Turning2WithSpraying
      R     "MAL1S019Par".Par.Switches1.StaOn11; // Turning2WithDosing

      L     "G145M".A_2311_MXZ41MA.Ma.OutPositionAngle;
      T     "G145M".A_2311_MXZ41MA.Ma.OutPositionAngle;

      L     "G145M".A_2311_MXZ41MA.Ma.OutPositionRel;
      T     "G145M".A_2311_MXZ41MA.Ma.OutPositionRel;

e603: NOP   0;
E603: NOP   0;


NETWORK
TITLE =ASW_6040: Set fanspeed by delta-t
//Die Drehzahl des Ventilators wird zwischen dem Rezeptsollwert, als Untere
//Grenze, und 100% oder Rezeptsollwert, als obere Grenze, geregelt. Die Regelung
//erfolgt nach folgendem Prinzip:
//"Delta-T" ist die Differenz zwischen der Soll-Temperatur (Rezeptsollwert) unter
//der Horde und der gemessenen Ist-Temperatur über der Horde.
//Steigt die Ist-Temperatur über der Horde und "Delta-T" wird > als der Sollwert
//im Rezept, so wird die Drehzahl des Ventilators stufenweise erhöht. Maximale
//Drehzahl ist 100% oder Rezeptsollwert.
//Sinkt die Ist-Temperatur über der Horde und "Delta-T" wird < als der Sollwert
//im
//Rezept, so wird die Drehzahl des Ventilators stufenweise verringert. Minimale
//Drehzahl ist der Rezeptsollwert.
//Die Rampen (Stufen) werden durch den Technologen festgelegt und in Programmcode
//eingetragen. Es sind keine Rezeptsollwerte.
      NOP   0;
//====>BRT070310
// recipe setpoint
//      L     "MAL1S019Par".StepAct.SpeedVentilatorBasic
//      L     0
//      ==I                               // no fan during turning
//      SPB   e604                        // JV040908
      AN(   ;
      A(    ;
      L     "MAL1S019Par".Par.ParIntMachine.ActualStep;
      L     1;
      ==I   ;
      )     ;
      AN(   ;
      L     "MAL1S019Par".Par.ProcessValue.StepTimeAct; // in ms
      L     L#1000; // in first secunde steptime
      >D    ;
      )     ;
      )     ;
// BRT070310 - berechneter Targetwert darf nur bei StepNr.1 oder! Rezeptwert-Änderung überschrieben werden
      A(    ;
      L     "MAL1S019Par".StepAct.SpeedVentilatorBasic;
      L     "MAL1S019Par".Par.ParIntProcess.Value23; // Rezeptwert vor Änderung
      ==D   ;
      )     ;
      JC    regu;
      L     "MAL1S019Par".StepAct.SpeedVentilatorBasic;
      T     "MAL1S019Par".Par.ParIntProcess.Value23; // Rezeptwert vor Änderung
      JU    Summ;
regu: NOP   0;

// BRT070310 - nicht nötig, da obige Änderung bei Änderung Rezeptwert (Modify) auch Target-Wert neu lädt
//      U     "MAL1S019".ToASW.CmdModify
//      SPB   Summ
//<====BRT070310

// Setpoint
      L     "MAL1S019Par".StepAct.TemperaturAboveFloor;
      L     "MAL1S019Par".StepAct.TemperaturBelowFloor;
      -D    ;
      T     "MAL1S019Par".Par.ProcessValue.SetpointDeltaTempDint;
// actual value
//10.04.17 donky. set average delta temperature regulating for testing purposes
      L     "G148M".A_2391_BTE02.OutValueUnits; //AIR TEMPERATURE ABOVE FLOOR
      L     "G148M".A_2391_BTE04.OutValueUnits; //AIR TEMPERATURE ABOVE FLOOR
      +D    ;
      DTR   ;
      L     2.000000e+000;
      /R    ;
      T     #tmpAverageTemp1;

      L     "G148M".A_2391_BTE01.OutValueUnits; //AIR TEMPERATURE BELOW FLOOR
      L     "G148M".A_2391_BTE03.OutValueUnits; //AIR TEMPERATURE BELOW FLOOR
      +D    ;
      DTR   ;
      L     2.000000e+000;
      /R    ;

      L     #tmpAverageTemp1;
      TAK   ;
      -R    ;
      TRUNC ;
      L     L#10; //BRT070310
      /D    ; //BRT070310

      T     "MAL1S019Par".Par.ProcessValue.ActValueDeltaTempDint;

// flags to inc/dec
      L     "MAL1S019Par".Par.ProcessValue.SetpointDeltaTempDint;
      -D    ;
      T     "MAL1S019Par".Par.ProcessValue.ResultDeltaTemp;
      L     L#0;
      >D    ;
      =     "MAL1S019Par".Par.FlagProcess1.DeltaTempPlus;
      <D    ;
      =     "MAL1S019Par".Par.FlagProcess1.DeltaTempMinus;

      A     "MAL1S019Par".Par.FlagProcess1.DeltaTempPlus;
//      U     "SYS_Scan0_Tick1min"
      A     "SYS_Scan0_Tick30s"; //Scan0_Tick30s
      JCN   dec;
      L     "MAL1S019Par".Par.ParIntMachine.TargetSpeedGermFan;
      L     100; // linmit max
      >=I   ;
      O(    ; //JV160710 =====>
      TAK   ;
      L     "MAL1S019Par".StepAct.SpeedVentilatorMaximal;
      >=I   ;
      A(    ;
      L     "MAL1S019Par".StepAct.SpeedVentilatorMaximal;
      L     "MAL1S019Par".StepAct.SpeedVentilatorBasic;
      >=I   ;
      )     ;
      )     ; //JV160710 <=====
      JC    dec;
      L     "MAL1S019Par".Par.ParIntMachine.TargetSpeedGermFan;
      L     1;
      +I    ;
      T     "MAL1S019Par".Par.ParIntMachine.TargetSpeedGermFan;
      JU    e604;
dec:  NOP   0;
      A     "MAL1S019Par".Par.FlagProcess1.DeltaTempMinus;
      O(    ; //JV160710 =====>
      L     "MAL1S019Par".Par.ParIntMachine.TargetSpeedGermFan;
      L     "MAL1S019Par".StepAct.SpeedVentilatorMaximal;
      >I    ;
      )     ; //JV160710 <=====
//      U     "SYS_Scan0_Tick1min"
      A     "SYS_Scan0_Tick30s"; //Scan0_Tick30s
      JCN   e604;
      L     "MAL1S019Par".Par.ParIntMachine.TargetSpeedGermFan;
      L     "MAL1S019Par".StepAct.SpeedVentilatorBasic; // linmit min
      <=I   ;
      JC    e604;
      L     "MAL1S019Par".Par.ParIntMachine.TargetSpeedGermFan;
      L     1;
      -I    ;
      T     "MAL1S019Par".Par.ParIntMachine.TargetSpeedGermFan;
      JU    e604;

Summ: NOP   0;
      L     "MAL1S019Par".StepAct.SpeedVentilatorBasic;
      T     "MAL1S019Par".Par.ParIntMachine.TargetSpeedGermFan;
      A     "MAL1S019Par".Par.FlagProcess.ProcessEnd; // JV030908
      AN    "MAL1S019".PCRead.Step.StEmptying;
      AN    "MAL1S019".PCRead.Step.StEmptied;
      JCN   e604;
      L     "MAL1S019Par".Par.ParIntProcess.SavedTargetSpeedGermFan;
      T     "MAL1S019Par".Par.ParIntMachine.TargetSpeedGermFan;
e604: NOP   0;
// store actual setpoint
      A     "MAL1S019Par".Par.FlagProcess.ProcessActive;
      A(    ;
      L     "MAL1S019Par".StepAct.SpeedVentilatorBasic;
      L     0; // setpoint recipe > 0
      >I    ;
      )     ;
      JCN   E604;
      L     "MAL1S019Par".StepAct.SpeedVentilatorBasic;
      T     "MAL1S019Par".Par.ParIntProcess.SavedTargetSpeedGermFan;
E604: NOP   0;
//-------------------------------------------------------------------------------------------------
//--- Ventilator 2 einzeln geregelt ---
      AN(   ;
      A(    ;
      L     "MAL1S019Par".Par.ParIntMachine.ActualStep;
      L     1;
      ==I   ;
      )     ;
      AN(   ;
      L     "MAL1S019Par".Par.ProcessValue.StepTimeAct; // in ms
      L     L#1000; // in first secunde steptime
      >D    ;
      )     ;
      )     ;
// BRT040310 - berechneter Targetwert darf nur bei StepNr.1 oder! Rezeptwert-Änderung überschrieben werden
      A(    ;
      L     "MAL1S019Par".StepAct.SpeedVentilatorBasic;
      L     "MAL1S019Par".Par.ParIntProcess.Value25; // Rezeptwert vor Änderung
      ==D   ;
      )     ;
      JC    reg1;
      L     "MAL1S019Par".StepAct.SpeedVentilatorBasic;
      T     "MAL1S019Par".Par.ParIntProcess.Value25; // Rezeptwert vor Änderung
      JU    Sum1;
reg1: NOP   0;
// Setpoint
      L     "MAL1S019Par".StepAct.TemperaturAboveFloor;
      L     "MAL1S019Par".StepAct.TemperaturBelowFloor;
      -D    ;
      T     "MAL1S019Par".Par.ProcessValue.Value13; // Setpoint Delta Temp
// actual value
//      L     "G148M".A_2391_BTE04.OutValueUnits    //AIR TEMPERATURE ABOVE FLOOR
//      L     "G148M".A_2391_BTE03.OutValueUnits    //AIR TEMPERATURE BELOW FLOOR
//      -D
//      L     L#10                        //BRT060310
//      /D                                //BRT060310

//10.04.17 donky. set average delta temperature regulating for testing purposes
      L     "MAL1S019Par".Par.ProcessValue.ActValueDeltaTempDint;
      T     "MAL1S019Par".Par.ProcessValue.Value14; // Actual Value Delta Temp

// flags to inc/dec
      L     "MAL1S019Par".Par.ProcessValue.Value13; // Setpoint Delta Temp
      -D    ;
      T     "MAL1S019Par".Par.ProcessValue.Value15; // Result Delta Temp
      L     L#0;
      >D    ;
      =     "MAL1S019Par".Par.FlagProcess1.Inf23; // Delta Temp Plus
      <D    ;
      =     "MAL1S019Par".Par.FlagProcess1.Inf24; // Delta Temp Minus

      A     "MAL1S019Par".Par.FlagProcess1.Inf23; // Delta Temp Plus
//BRT203010      U     "SYS_Scan0_Tick1min"
      A     "SYS_Scan0_Tick30s"; //Scan0_Tick30s
      JCN   dec1;
      L     "MAL1S019Par".Par.ParIntProcess.Value26; // Target Speed GermFan 2
      L     100; // linmit max
      >=I   ;
      O(    ; //JV160710 =====>
      TAK   ;
      L     "MAL1S019Par".StepAct.SpeedVentilatorMaximal;
      >=I   ;
      A(    ;
      L     "MAL1S019Par".StepAct.SpeedVentilatorMaximal;
      L     "MAL1S019Par".StepAct.SpeedVentilatorBasic;
      >=I   ;
      )     ;
      )     ; //JV160710 <=====
      JC    dec1;
      L     "MAL1S019Par".Par.ParIntProcess.Value26; // Target Speed GermFan 2
      L     1;
      +I    ;
      T     "MAL1S019Par".Par.ParIntProcess.Value26; // Target Speed GermFan 2
      JU    e614;
dec1: NOP   0;
      A     "MAL1S019Par".Par.FlagProcess1.Inf24; // Delta Temp Minus
      O(    ; //JV160710 =====>
      L     "MAL1S019Par".Par.ParIntProcess.Value26;
      L     "MAL1S019Par".StepAct.SpeedVentilatorMaximal;
      >I    ;
      )     ; //JV160710 <=====
//BRT200310      U     "SYS_Scan0_Tick1min"
      A     "SYS_Scan0_Tick30s"; //Scan0_Tick30s
      JCN   e614;
      L     "MAL1S019Par".Par.ParIntProcess.Value26; // Target Speed GermFan 2
      L     "MAL1S019Par".StepAct.SpeedVentilatorBasic; // linmit min
      <=I   ;
      JC    e614;
      L     "MAL1S019Par".Par.ParIntProcess.Value26; // Target Speed GermFan 2
      L     1;
      -I    ;
      T     "MAL1S019Par".Par.ParIntProcess.Value26; // Target Speed GermFan 2
      JU    e614;

Sum1: NOP   0;
      L     "MAL1S019Par".StepAct.SpeedVentilatorBasic;
      T     "MAL1S019Par".Par.ParIntProcess.Value26; // Target Speed GermFan 2
      A     "MAL1S019Par".Par.FlagProcess.ProcessEnd; // JV030908
      AN    "MAL1S019".PCRead.Step.StEmptying;
      AN    "MAL1S019".PCRead.Step.StEmptied;
      JCN   e614;
      L     "MAL1S019Par".Par.ParIntProcess.Value27; // Saved Target Speed GermFan 2
      T     "MAL1S019Par".Par.ParIntProcess.Value26; // Target Speed GermFan 2
e614: NOP   0;
// store actual setpoint
      A     "MAL1S019Par".Par.FlagProcess.ProcessActive;
      A(    ;
      L     "MAL1S019Par".StepAct.SpeedVentilatorBasic;
      L     0; // setpoint recipe > 0
      >I    ;
      )     ;
      JCN   E614;
      L     "MAL1S019Par".StepAct.SpeedVentilatorBasic;
      T     "MAL1S019Par".Par.ParIntProcess.Value27; // Saved Target Speed GermFan 2
E614: NOP   0;

NETWORK
TITLE =ASW_6050: Position waste air
//Der Betriebsart Sommerbetrieb/Winterbetrieb wird durch den Bediener per Rezept
//bestimmt.
//Wird die Kühlung im Rezept angewählt, so erfolgt die Umschaltung AUF
//Sommerbetrieb. Die Frischluftklappe wird nach dem Rezeptsollwert gestellt.
//Es erfolgt keine Regelung.
//Wird die Kühlung im Rezept abgewählt, so erfolgt die Umschaltung AUF
//Winterbetrieb. Die Frischluftklappe wird zuerst nach dem Rezeptsollwert
//gestellt. Der Rezeptsollwert ist die untere Grenze für die Regelung.
//Wird die Soll-Temperatur unter der Horde von Kühl- Heizanlage nicht eingehalten
//-Temperatur zu hoch und der Schaltpunkt überschritten, so wird die
//Frischluftklappe stufenweise geöffnet.
//Maximalwert ist 100%.
//Wird die Soll-Temperatur unter der Horde von Kühl- Heizanlage nicht eingehalten
//-Temperatur zu niedrig und der Schaltpunkt unterschritten, so wird die
//Frischluftklappe stufenweise geschlossen.
//Minimalwert ist der Rezeptsollwert.
//--------------------------------------------------------------------------------
//      NOP   0
//// setpoint waste air                    = 100% - setpoint fresh air
//      L     100
//      L     "MAL1S019Par".StepAct.PosFreshAirFlapBasic
//      -I
//      T     "MAL1S019Par".StepAct.PosWasteAirFlapBasic
//
//// setpoint limit maximal position fresh air
//      L     100
//      T     "MAL1S019Par".StepAct.PosFreshAirFlapMax    // limit max
//      L     L#10                        // 1,0°
//      T     "MAL1S019Par".StepAct.DeltaTempSwitchpointAir
//
//// recipe setpoint
//      L     "MAL1S019Par".Par.ProcessValue.StepTimeAct    // in ms
//      L     L#1000                      // in first secunde steptime
//      >D
//      SPB   Reg
//      SPA   summ
//Reg:  NOP   0
//
//// Cooling or heating from cooling defive active --> no flap regulation!
////      U     "ENG_RemarkFlag"
////      U     "ComDB_Cooling".Ma.ACK.ActivFlag.Cool.Germinating_1_Started //
//Internal or external coooling is running
////      O     "MAL1S017".ToASW.CmdModify
////      SPB   summ
//
////Conditions to activate cooling -- With flap regulation
//      U(
//      L     1
//      L     "MAL1S019Par".StepAct.Cooling    // On/Off
//      ==I                               // Cooling on
//      U     "MAL1S019Par".Par.FlagProcess.ProcessActive
//      )
//      U     "G150M".A_2360_MXZ01.StStartedFwd
//      U     "G150M".A_2360_MXZ02.StStartedFwd
//      U(
//      L     "G269M".A_3191_BTE11.OutValueUnits    //WET BULB TEMPERATURE OUTSIDE
//      L     20                          // 2,0°C Hysteresis
//      -D
//      L     "MAL1S019Par".StepAct.TemperaturBelowFloor    //SET POINT
//TEMPERATURE RECIPE
//      >=D
//      )
//      U(
//      L     "G148M".A_2391_BTE01.OutValueUnits    //AIR TEMPERATURE BELOW FLOOR
//GM2
//      L     10                          // 1,0°C Hysteresis
//      -D
//      L     "MAL1S019Par".StepAct.TemperaturBelowFloor    //SET POINT
//TEMPERATURE RECIPE
//      >=D
//      )
//      U(
//      L     "G148M".A_2391_BTE02.OutValueUnits    //AIR TEMPERATURE ABOVE FLOOR
//GM2
//      L     20                          // 2,0°C Hysteresis
//      -D
//      L     "MAL1S019Par".StepAct.TemperaturBelowFloor    //SET POINT
//TEMPERATURE RECIPE
//      >=D
//      )
//      S     "MAL1S019Par".Par.FlagProcess.Cooling_Activ
//
//      U(
//      L     0
//      L     "MAL1S019Par".StepAct.Cooling    // On/Off
//      ==I                               // Cooling off
//      )
//      ON    "G150M".A_2360_MXZ01.StStartedFwd
//      ON    "G150M".A_2360_MXZ02.StStartedFwd
//      O(
//      L     "G269M".A_3191_BTE11.OutValueUnits    //WET BULB TEMPERATURE OUTSIDE
//      L     10                          // 1,0°C Hysteresis
//      +D
//      L     "MAL1S019Par".StepAct.TemperaturBelowFloor    //SET POINT
//TEMPERATURE RECIPE
//      <D
//      )
//      O(
//      L     "G148M".A_2391_BTE02.OutValueUnits    //AIR TEMPERATURE ABOVE FLOOR
//GM1
//      L     10                          // 1,0°C Hysteresis
//      +D
//      L     "MAL1S019Par".StepAct.TemperaturBelowFloor    //SET POINT
//TEMPERATURE RECIPE
//      <D
//      )
//      R     "MAL1S019Par".Par.FlagProcess.Cooling_Activ
//
//      U     "MAL1S019Par".Par.FlagProcess.Cooling_Activ
//      SPB   summ
//
//// Check the minimum opening of fresh air louver
//      U(
//      L     "MAL1S019Par".Par.ParIntMachine.TargetPosFreshAir
//      L     "MAL1S019Par".StepAct.PosFreshAirFlapBasic
//      <I
//      )
//      SPBN  modi
//      L     "MAL1S019Par".StepAct.PosFreshAirFlapBasic    //Basic position %
//      T     "MAL1S019Par".Par.ParIntMachine.TargetPosFreshAir
//modi: NOP   0
//
////-Recipe modify-
//      U(                                // Nach gesundem Menschenverstand
//      L     "MAL1S019Par".StepAct.PosFreshAirFlapBasic
//      L     "MAL1S019Par".Par.ParIntMachine.TargetPosFreshAir
//      >I
//      U     "MAL1S019Par".Par.FlagProcess1.FreshAirFlapOPEN
//      )
//      O(                                // Nach gesundem Menschenverstand
//      L     "MAL1S019Par".StepAct.PosFreshAirFlapBasic
//      L     "MAL1S019Par".Par.ParIntMachine.TargetPosFreshAir
//      <I
//      U     "MAL1S019Par".Par.FlagProcess1.FreshAirFlapCLOSE
//      )
//      O(                                // Nach gesundem Menschenverstand
//      L     "MAL1S019Par".StepAct.PosFreshAirFlapBasic
//      L     "MAL1S019Par".Par.ParIntMachine.TargetPosFreshAir
//      <>I
//      UN    "MAL1S019Par".Par.FlagProcess1.FreshAirFlapOPEN
//      UN    "MAL1S019Par".Par.FlagProcess1.FreshAirFlapCLOSE
//      )
//      O(                                // 1. Versuch den Technologen ruhig
//stellen
//      L     "MAL1S019Par".StepAct.PosFreshAirFlapBasic
//      L     "MAL1S019Par".Par.ParIntProcess.SavedTargetPosFreshAir
//      <>I
//      )
//      U     "MAL1S019".ToASW.CmdModify
//      SPB   summ
////      L     "G148M".A_2391_BTE01.OutValueUnits    //AIR TEMPERATURE BELOW
//FLOOR
////      L     L#10                        // von xx,xx°C AUF xx,x°C
////      /D
////      L     "MAL1S017Par".StepAct.TemperaturBelowFloor
////      -D
////      L     "MAL1S017Par".StepAct.DeltaTempSwitchpointAir
////      >D
////      =     "MAL1S017Par".Par.FlagProcess1.FreshAirFlapOPEN
//
////      L     "G128M".A_2191_BTE01.OutValueUnits    //AIR TEMPERATURE BELOW
//FLOOR
////      L     L#10                        // von xxx,xx°C AUF xxx,x°C
////      /D
////      L     "MAL1S017Par".StepAct.TemperaturBelowFloor
////      TAK
////      -D
////      L     "MAL1S017Par".StepAct.DeltaTempSwitchpointAir
////      >D
////      =     "MAL1S017Par".Par.FlagProcess1.FreshAirFlapCLOSE
//      U(
//      L     "G148M".A_2391_BTE01.OutValueUnits    //AIR TEMPERATURE BELOW FLOOR
//GM1
//      L     "MAL1S019Par".StepAct.TemperaturBelowFloor    //SET POINT
//TEMPERATURE RECIPE
//      <D
//      )
//      U(
//      L     "G269M".A_3191_BTE11.OutValueUnits    //WET BULB TEMPERATURE OUTSIDE
//      L     "G148M".A_2391_BTE02.OutValueUnits    //AIR TEMPERATURE ABOVE FLOOR
//GM1
//      >D
//      )
//      O
//      U(
//      L     "G148M".A_2391_BTE01.OutValueUnits    //AIR TEMPERATURE BELOW FLOOR
//GM1
//      L     "MAL1S019Par".StepAct.TemperaturBelowFloor    //SET POINT
//TEMPERATURE RECIPE
//      >D
//      )
//      U(
//      L     "G269M".A_3191_BTE11.OutValueUnits    //WET BULB TEMPERATURE OUTSIDE
//      L     "G148M".A_2391_BTE01.OutValueUnits    //AIR TEMPERATURE BELOW FLOOR
//GM1
//      <D
//      )
//      =     "MAL1S019Par".Par.FlagProcess1.FreshAirFlapOPEN
//
//      U(
//      L     "G148M".A_2391_BTE01.OutValueUnits    //AIR TEMPERATURE BELOW FLOOR
//GM1
//      L     "MAL1S019Par".StepAct.TemperaturBelowFloor    //SET POINT
//TEMPERATURE RECIPE
//      <D
//      )
//      U(
//      L     "G269M".A_3191_BTE11.OutValueUnits    //WET BULB TEMPERATURE OUTSIDE
//      L     "G148M".A_2391_BTE02.OutValueUnits    //AIR TEMPERATURE ABOVE FLOOR
//GM1
//      <D
//      )
//      =     "MAL1S019Par".Par.FlagProcess1.FreshAirFlapCLOSE
//
//      U     "MAL1S019Par".Par.FlagProcess1.FreshAirFlapOPEN
//      U     "SYS_Scan0_Tick1min"
//      SPBN  dez
//      L     "MAL1S019Par".Par.ParIntMachine.TargetPosWasteAir
//      L     100                         // limit max
//      >=I
//      SPB   dez
//      L     "MAL1S019Par".Par.ParIntMachine.TargetPosWasteAir
//      L     1
//      +I
//      T     "MAL1S019Par".Par.ParIntMachine.TargetPosWasteAir
//      SPA   e605
//dez:  NOP   0
//      U     "MAL1S019Par".Par.FlagProcess1.FreshAirFlapCLOSE
//      U     "SYS_Scan0_Tick1min"
//      SPBN  e605
//      L     "MAL1S019Par".Par.ParIntMachine.TargetPosWasteAir
//      L     "MAL1S019Par".StepAct.PosFreshAirFlapBasic    // limit min
//      <=I
//      SPB   e605
//      L     "MAL1S019Par".Par.ParIntMachine.TargetPosWasteAir
//      L     1
//      -I
//      T     "MAL1S019Par".Par.ParIntMachine.TargetPosWasteAir
//      SPA   e605
//
//summ: NOP   0
//      U     "G269M".read_3191
//      SPBN  bypa
//      U(
//      L     "G148M".A_2391_BTE02.OutValueUnits    //AIR TEMPERATURE ABOVE FLOOR
//GM1
//      L     10                          // 1,0°C Hysteresis
//      -D
//      L     "G269M".A_3191_BTE11.OutValueUnits    //WET BULB TEMPERATURE OUTSIDE
//      >=D
//      )
//      SPB   tar1
//      U(
//      L     "G148M".A_2391_BTE02.OutValueUnits    //AIR TEMPERATURE ABOVE FLOOR
//GM1
//      L     10                          // 1,0°C Hysteresis
//      +D
//      L     "G269M".A_3191_BTE11.OutValueUnits    //WET BULB TEMPERATURE OUTSIDE
//      <=D
//      )
//      SPB   tar0
//      SPA   bypa
//tar1: L     100                         //open fresh air 100%
//      T     "MAL1S019Par".Par.ParIntMachine.TargetPosFreshAir
//      SPA   bypa
//tar0: L     "MAL1S019Par".StepAct.PosFreshAirFlapBasic    //close fresh air to
//Basic position %
//      T     "MAL1S019Par".Par.ParIntMachine.TargetPosFreshAir
//bypa: NOP   0
////************************************************************************
//      U     "MAL1S019Par".Par.FlagProcess.ProcessEnd    // JV030908
//      UN    "MAL1S019".PCRead.Step.StEmptying
//      UN    "MAL1S019".PCRead.Step.StEmptied    // JV030908
//      SPBN  e605
//      L     "MAL1S019Par".Par.ParIntProcess.SavedTargetPosFreshAir
//      T     "MAL1S019Par".Par.ParIntMachine.TargetPosFreshAir
//e605: NOP   0
//      L     100
//      L     "MAL1S019Par".Par.ParIntMachine.TargetPosFreshAir
//      -I
//      T     "MAL1S019Par".Par.ParIntMachine.TargetPosWasteAir
//// store actual setpoint
//      U     "MAL1S019Par".Par.FlagProcess.ProcessActive
//      U(
//      L     "MAL1S019Par".StepAct.PosFreshAirFlapBasic
//      L     0                           // setpoint recipe > 0
//      >I
//      )
//      SPBN  E605
//      L     "MAL1S019Par".StepAct.PosFreshAirFlapBasic
//      T     "MAL1S019Par".Par.ParIntProcess.SavedTargetPosFreshAir
//E605: NOP   0
//
//BRT070310 - keine AMBEV Steuerung!!!
      NOP   0;
// setpoint limit maximal position fresh air
      L     100;
      T     "MAL1S019Par".StepAct.PosFreshAirFlapMax; // limit max
      L     L#5; // 0,5°
      T     "MAL1S019Par".StepAct.DeltaTempSwitchpointAir;

// recipe setpoint
      AN(   ;
      A(    ;
      L     "MAL1S019Par".Par.ParIntMachine.ActualStep;
      L     1;
      ==I   ;
      )     ;
      AN(   ;
      L     "MAL1S019Par".Par.ProcessValue.StepTimeAct; // in ms
      L     L#1000; // in first secunde steptime
      >D    ;
      )     ;
      )     ;
// BRT17102009 - berechneter Targetwert darf nur bei StepNr.1 oder! Rezeptwert-Änderung überschrieben werden
      A(    ;
      L     "MAL1S019Par".StepAct.PosFreshAirFlapBasic;
      L     "MAL1S019Par".Par.ParIntProcess.Value24; // Rezeptwert vor Änderung
      ==D   ;
      )     ;
      JC    Reg;
      L     "MAL1S019Par".StepAct.PosFreshAirFlapBasic;
      T     "MAL1S019Par".Par.ParIntProcess.Value24; // Rezeptwert vor Änderung

      L     "MAL1S019Par".StepAct.PosFreshAirFlapBasic;
      T     "MAL1S019Par".Par.ParIntMachine.TargetPosFreshAir;
      JU    e605;
Reg:  NOP   0;

// Cooling or heating from cooling defive active --> no flap regulation!
//BRT030310 - Cooling angewählt in Rezept!
      A     "MAL1S019Par".Par.FlagProcess.Cooling; // request cooling
      JC    summ;
//=> 17.02.2018 donky. deleted by new flaps release
//      L     "G148M".A_2391_BTE01.OutValueUnits    //AIR TEMPERATURE BELOW FLOOR
//      L     L#10                        // von xx,xx°C AUF xx,x°C
//      /D
//      L     "MAL1S019Par".StepAct.TemperaturBelowFloor
//      -D
//      L     "MAL1S019Par".StepAct.DeltaTempSwitchpointAir
//      >D
//      =     "MAL1S019Par".Par.FlagProcess1.FreshAirFlapOPEN

//      L     "G148M".A_2391_BTE01.OutValueUnits    //AIR TEMPERATURE BELOW FLOOR
//      L     L#10                        // von xxx,xx°C AUF xxx,x°C
//      /D
//      L     "MAL1S019Par".StepAct.TemperaturBelowFloor
//      TAK
//      -D
//      L     "MAL1S019Par".StepAct.DeltaTempSwitchpointAir
//      >D
//      =     "MAL1S019Par".Par.FlagProcess1.FreshAirFlapCLOSE

//      A     "MAL1S019Par".Par.FlagProcess1.FreshAirFlapOPEN
//      A     "SYS_Scan0_Tick1min"
//      JCN   dez
//      L     "MAL1S019Par".Par.ParIntMachine.TargetPosFreshAir
//      L     "MAL1S019Par".StepAct.PosFreshAirFlapMax    // limit max
//      >=I
//      JC    dez
//      L     "MAL1S019Par".Par.ParIntMachine.TargetPosFreshAir
//      L     1
//      +I
//      T     "MAL1S019Par".Par.ParIntMachine.TargetPosFreshAir
//      JU    e605
//dez:  NOP   0
//      A     "MAL1S019Par".Par.FlagProcess1.FreshAirFlapCLOSE
//      A     "SYS_Scan0_Tick1min"
//      JCN   e605
//      L     "MAL1S019Par".Par.ParIntMachine.TargetPosFreshAir
//      L     "MAL1S019Par".StepAct.PosFreshAirFlapBasic    // limit min
//      <=I
//      JC    e605
//      L     "MAL1S019Par".Par.ParIntMachine.TargetPosFreshAir
//      L     1
//      -I
//      T     "MAL1S019Par".Par.ParIntMachine.TargetPosFreshAir
//      JU    e605
//<=
      AN    "MAL1S019Par".Par.FlagProcess.ProcessActive;
      JC    e605;
      L     "RegDBKK3_1".LMN;
      TRUNC ;
      T     "MAL1S019Par".Par.ParIntMachine.TargetPosFreshAir;
      JU    e605;
summ: NOP   0;
      L     "MAL1S019Par".StepAct.PosFreshAirFlapBasic;
      T     "MAL1S019Par".Par.ParIntMachine.TargetPosFreshAir;
      JU    e605;

e605: NOP   0;
//------------------------------------------------------------------------------------------------
//--- Position Fresh-/Recycling-Air Flap 2 ---
// recipe setpoint
      AN(   ;
      A(    ;
      L     "MAL1S019Par".Par.ParIntMachine.ActualStep;
      L     1;
      ==I   ;
      )     ;
      AN(   ;
      L     "MAL1S019Par".Par.ProcessValue.StepTimeAct; // in ms
      L     L#1000; // in first secunde steptime
      >D    ;
      )     ;
      )     ;
// BRT17102009 - berechneter Targetwert darf nur bei StepNr.1 oder! Rezeptwert-Änderung überschrieben werden
      A(    ;
      L     "MAL1S019Par".StepAct.PosFreshAirFlapBasic;
      L     "MAL1S019Par".Par.ParIntProcess.Value28; // Rezeptwert vor Änderung
      ==D   ;
      )     ;
      JC    Reg1;
      L     "MAL1S019Par".StepAct.PosFreshAirFlapBasic;
      T     "MAL1S019Par".Par.ParIntProcess.Value28; // Rezeptwert vor Änderung

      L     "MAL1S019Par".StepAct.PosFreshAirFlapBasic;
      T     "MAL1S019Par".Par.ParIntProcess.Value29; // Target Position FreshAir 2
      JU    e615;
Reg1: NOP   0;

// Cooling or heating from cooling defive active --> no flap regulation!
//BRT030310 - Cooling angewählt in Rezept!
      A     "MAL1S019Par".Par.FlagProcess.Cooling; // request cooling
      JC    sum1;
//=> 17.02.2018 donky. deleted by new flaps release
//      L     "G148M".A_2391_BTE03.OutValueUnits    //AIR TEMPERATURE BELOW FLOOR
//      L     L#10                        // von xx,xx°C AUF xx,x°C
//      /D
//      L     "MAL1S019Par".StepAct.TemperaturBelowFloor
//      -D
//      L     "MAL1S019Par".StepAct.DeltaTempSwitchpointAir
//      >D
//      =     "MAL1S019Par".Par.FlagProcess.Inf05    // FreshAir Flap OPEN

//      L     "G148M".A_2391_BTE03.OutValueUnits    //AIR TEMPERATURE BELOW FLOOR
//      L     L#10                        // von xxx,xx°C AUF xxx,x°C
//      /D
//      L     "MAL1S019Par".StepAct.TemperaturBelowFloor
//      TAK
//      -D
//      L     "MAL1S019Par".StepAct.DeltaTempSwitchpointAir
//      >D
//      =     "MAL1S019Par".Par.FlagProcess.Inf06    // FreshAir Flap CLOSE

//      A     "MAL1S019Par".Par.FlagProcess.Inf05    // FreshAir Flap OPEN
//      A     "SYS_Scan0_Tick1min"
//      JCN   dez1
//      L     "MAL1S019Par".Par.ParIntProcess.Value29    // Target Position FreshAir 2
//      L     "MAL1S019Par".StepAct.PosFreshAirFlapMax    // limit max
//      >=I
//      JC    dez1
//      L     "MAL1S019Par".Par.ParIntProcess.Value29    // Target Position FreshAir 2
//      L     1
//      +I
//      T     "MAL1S019Par".Par.ParIntProcess.Value29    // Target Position FreshAir 2
//      JU    e615
//dez1: NOP   0
//      A     "MAL1S019Par".Par.FlagProcess.Inf06    // FreshAir Flap CLOSE
//      A     "SYS_Scan0_Tick1min"
//      JCN   e615
//      L     "MAL1S019Par".Par.ParIntProcess.Value29    // Target Position FreshAir 2
//      L     "MAL1S019Par".StepAct.PosFreshAirFlapBasic    // limit min
//      <=I
//      JC    e615
//      L     "MAL1S019Par".Par.ParIntProcess.Value29    // Target Position FreshAir 2
//      L     1
//      -I
//      T     "MAL1S019Par".Par.ParIntProcess.Value29    // Target Position FreshAir 2
//      JU    e615
//<=
      AN    "MAL1S019Par".Par.FlagProcess.ProcessActive;
      JC    e615;
      L     "RegDBKK3_2".LMN;
      TRUNC ;
      T     "MAL1S019Par".Par.ParIntProcess.Value29;
      JU    e615;

sum1: NOP   0;
      L     "MAL1S019Par".StepAct.PosFreshAirFlapBasic;
      T     "MAL1S019Par".Par.ParIntProcess.Value29; // Target Position FreshAir 2
      JU    e615;

e615: NOP   0;

NETWORK
TITLE =ASW_6080: Processtime Germinating
//      CALL  "SSA_MH_ProcessTime_Fct" , DB1017
//       InfDataReady :="MAL1S019".ToASW.InfDataReady
//       ProzessActive:="MAL1S017Par".Par.FlagProcess.ProcessActive
//       InStartTime  :="MAL1S017Par".Prozesstime.Starttime
//       OutStartTime :="MAL1S017Par".Prozesstime.Starttime
//       ProcessTime  :="MAL1S017Par".Prozesstime
//
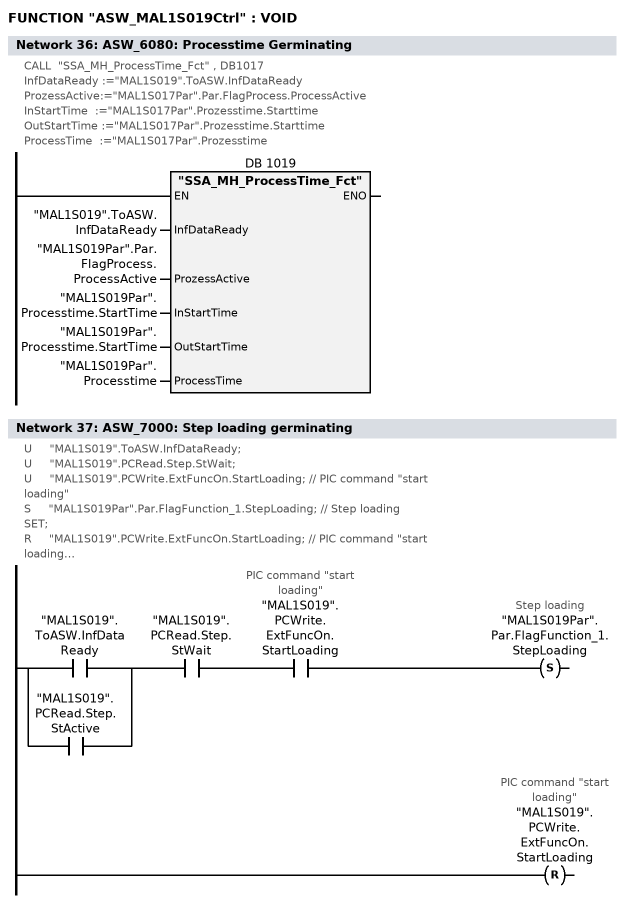
      CALL "SSA_MH_ProcessTime_Fct" , DB  1019 (
           InfDataReady             := "MAL1S019".ToASW.InfDataReady,
           ProzessActive            := "MAL1S019Par".Par.FlagProcess.ProcessActive,
           InStartTime              := "MAL1S019Par".Processtime.StartTime,
           OutStartTime             := "MAL1S019Par".Processtime.StartTime,
           ProcessTime              := "MAL1S019Par".Processtime);

NETWORK
TITLE =ASW_7000: Step loading germinating
//      U     "MAL1S019".ToASW.InfDataReady;
//      U     "MAL1S019".PCRead.Step.StWait;
//      U     "MAL1S019".PCWrite.ExtFuncOn.StartLoading; // PIC command "start
//loading"
//      S     "MAL1S019Par".Par.FlagFunction_1.StepLoading; // Step loading
//      SET;
//      R     "MAL1S019".PCWrite.ExtFuncOn.StartLoading; // PIC command "start
//loading"
////
//
//      L     WinCoS_BIW01_09PLC1BIW01_02.Ma.OutPositionAngle;
//      L     3600; // 360,0°
//      >=I   ;
//      U     "MAL1S019".ToASW.InfDataReady;
//      U     "MAL1S019".PCRead.Step.StActive;
//      U     "MAL1S019Par".Par.FlagFunction_1.StepLoading; // Step loading
//      =     "MAL1S019Par".Par.FlagFunction_1.LoadFirstPartEnd;
//
//      U     "MAL1S019".ToASW.InfDataReady;
//      U     "MAL1S019".PCRead.Step.StActive;
//      U     "MAL1S019Par".Par.FlagFunction_1.StepLoading; // Step loading
//      SPBN  E700;
//      L     "MAL1S019Par".RecipeHeader.Loading.LiftingPositionRound_1;
//      T     "MAL1S019Par".Par.ParIntProcess.NextLevelLoading; // next level
//
//      U(    ;
//      L     WinCoS_BIW01_09PLC1BIW01_02.Ma.OutPositionAngle;
//      L     "MAL1S019Par".Par.ParIntProcess.NextLevelLoading; // next level
//      >=I   ;
//      )     ;
//      O     "MAL1S019Par".Par.FlagMachine_0.Speed2ndRound;
//      SPB   Rnd2;
//      L     "MAL1S019Par".RecipeHeader.Loading.LoadingLevelRound_1;
//      T     "MAL1S019Par".Par.MachineValue.SOLLWERT_HUBZUG1_HOEHE;
//      T     "MAL1S019Par".Par.MachineValue.SOLLWERT_HUBZUG2_HOEHE;
//
//      L     "MAL1S019Par".RecipeHeader.Loading.LoadingSpeed_1;
//      T     "MAL1S019Par".Par.MachineValue.SollwertFahrantrieb;
//
//      SPA   Rnd1;
//Rnd2: NOP   0;
//      L     "MAL1S019Par".RecipeHeader.Loading.LoadingLevelRound_2;
//      T     "MAL1S019Par".Par.MachineValue.SOLLWERT_HUBZUG1_HOEHE;
//      T     "MAL1S019Par".Par.MachineValue.SOLLWERT_HUBZUG2_HOEHE;
//      L     10;
//      T     WinCoS_BIW01_09PLC1BIW01_02.Ma.Par.ParTolPosition;
//
//      L     15; // 15Hz = Wendegeschwindigkeit
//      T     "MAL1S019Par".Par.MachineValue.SollwertFahrantrieb;
//
//// Sicherheitsbit; damit bei manueller Rückwärtsfahrt über die 346°-Marke,
//nicht mit Loading Speed_0 durch den gefüllten KK gefahren wird!!
//      SET   ;
//      S     "MAL1S019Par".Par.FlagMachine_0.Speed2ndRound;
//
//Rnd1: NOP   0;
//      U  M 50.0;
//      =  M 50.0;
//      L     "MAL1S019Par".Par.ParIntMachine.TargetPosTravDriveLoad; // 450 = end
//position loading
//      T     WinCoS_BIW01_09PLC1BIW01_02.Ma.InPositionTarget;
//E700: NOP   0;

      A     "MAL1S019".ToASW.InfDataReady;
      O     "MAL1S019".PCRead.Step.StActive;
      A     "MAL1S019".PCRead.Step.StWait;
      A     "MAL1S019".PCWrite.ExtFuncOn.StartLoading; // PIC command "start loading"
      S     "MAL1S019Par".Par.FlagFunction_1.StepLoading; // Step loading
      SET   ;
      R     "MAL1S019".PCWrite.ExtFuncOn.StartLoading; // PIC command "start loading"
//
      NOP   0;


NETWORK
TITLE =Sub 7010: Germination loading finished
//      U     "MAL1S019".ToASW.InfDataReady;
//      U     "MAL1S019".PCRead.Step.StActive;
//
//      UN    "MAL1S019".ToASW.InfSameJobPrevSec;
//      UN    "MAL1S019".PCRead.Step.StEmptying; // steep 1
//      U     "MAL1S019".PCWrite.ExtFuncOn.FinishLoading; // PIC command "finish l
//oading"
//      U     "MAL1S019Par".Par.FlagFunction_1.StepLoading; // Step loading
//      S     "MAL1S019Par".Par.FlagFunction_1.FinishLoading; // loading is
//finished start process germinating
//      R     "MAL1S019Par".Par.FlagFunction_1.StepLoading; // Step loading
//
//      U     "MAL1S019".PCWrite.ExtFuncOn.FinishLoading; // PIC command "finish
//loading"
//      R     "MAL1S019".PCWrite.ExtFuncOn.FinishLoading; // PIC command "finish
//loading"
//
//      U     "MAL1S019Par".Par.FlagFunction_1.StepLoading; // Step loading
//      UN    "MAL1S019Par".Par.FlagFunction_1.FinishLoading; // loading is
//finished start process germinating
//      SPBN  save;
//      L     WinCoS_BIW01_09PLC1BIW01_02.Ma.OutPositionLeft;
//      L     WinCoS_BIW01_09PLC1BIW01_02.Ma.OutPositionRight;
//      +I    ;
//      L     2;
//      /I    ;
//      T     "MAL1S019Par".Par.ParIntMachine.LastLoadingLevel; // saved loading
//value
//save: NOP   0;
//
//      U     "MAL1S019".PCRead.Step.StReady;
//      O     "MAL1S019".PCRead.Step.StActive;
//      U     "MAL1S019Par".Par.FlagFunction_1.FinishLoading; // loading is
//finished start process germinating
//      UN     "MAL1S019Par".Par.FlagFunction_1.StepLoading; // Step loading
//      R     "MAL1S019Par".Par.FlagMachine_0.Speed2ndRound;
//fin:  NOP   0;
//E701: NOP   0;
// Previous Section always the Sec.801
///
      L     "MAL1S019".ToSSW.InPrevSecDB;
      L     0;
      <>I   ;
      JC    prev;
      L     801;
      T     "MAL1S019".ToSSW.InPrevSecDB;
prev: NOP   0;


      A     "MAL1S019".ToASW.InfDataReady;
      A     "MAL1S019".PCRead.Step.StActive;
      AN    "MAL1S019".PCRead.Step.StEmptying; //
      A     "MAL1S019".PCWrite.ExtFuncOn.FinishLoading; // PIC command "finish loading"
      A     "MAL1S019Par".Par.FlagFunction_1.StepLoading; // Step loading
      O(    ;
      AN    "MAL1S019".SecNom.Par1On.Cmd01; // With Loading
      AN    "MAL1S019".ToASW.InfSameBatchPrevSec;
      A     "MAL1S019".ToASW.InfDataReady;
      A     "MAL1S019".PCRead.Step.StActive;
      )     ;
      S     "MAL1S019Par".Par.FlagFunction_1.FinishLoading; // loading is finished start process germinating
      R     "MAL1S019Par".Par.FlagFunction_1.StepLoading; // Step loading

      A     "MAL1S019".PCWrite.ExtFuncOn.FinishLoading; // PIC command "finish loading"
      R     "MAL1S019".PCWrite.ExtFuncOn.FinishLoading; // PIC command "finish loading"


      A     "MAL1S019".PCRead.Step.StReady;
      O     "MAL1S019".PCRead.Step.StActive;
      A     "MAL1S019Par".Par.FlagFunction_1.FinishLoading; // loading is finished start process germinating
      AN    "MAL1S019Par".Par.FlagFunction_1.StepLoading; // Step loading
      R     "MAL1S019Par".Par.FlagMachine_0.Speed2ndRound;
      NOP   0;
      NOP   0;


NETWORK
TITLE =ASW_8000:  Step unloading germination


      A     "MAL1S019".ToASW.InfDataReady;
      A     "MAL1S019".PCRead.Step.StEmptying;
//====>BRT070310
      A(    ;
      O     "MAL1S019".ToASW.InfSameJobNextSec;
      O(    ;
      L     831; // Next Section: MAL1S031
      L     "MAL1S019".SecNom.HEADER.Kilning_vessel_1; // Target in recipe
      ==I   ;
      )     ;
      )     ;
//<====BRT070310
      AN    "MAL1S019Par".Par.FlagFunction_1.StepUnloading; // Step unloading
      AN    "MAL1S019Par".Par.FlagFunction_1.FinishUnloading;
      A     "MAL1S019Par".Par.FlagMachine_0.CouplingDischargFinished;
      A     "MAL1S019Par".Par.FlagMachine_0.WallUnCoupled;
//BRT070310 - Start Unloading Button vergessen
      A     "MAL1S019".PCWrite.ExtFuncOn.StartUnLoading; // PIC command "Start Unloading"
      S     "MAL1S019Par".Par.FlagFunction_1.StepUnloading; // Step unloading

//BRT070310 - Start Unloading Button vergessen
      A     "MAL1S019".PCWrite.ExtFuncOn.StartUnLoading; // PIC command "Start Unloading"
      R     "MAL1S019".PCWrite.ExtFuncOn.StartUnLoading; // PIC command "Start Unloading"


      A     "MAL1S019Par".Par.FlagFunction_1.StepUnloading; // Step unloading
      A     "MAL1S019Par".Par.FlagFunction_1.UnloadingStarted;
//====>BRT070310
      A(    ;
      O     "MAL1S019".ToASW.spare34; // infNextSectionFeeding
      O(    ;
      L     831; // Next Section: MAL1S031
      L     "MAL1S019".SecNom.HEADER.Kilning_vessel_1; // Target in recipe
      ==I   ;
      )     ;
      )     ;
//<====BRT070310
      =     "MAL1S019Par".Par.FlagFunction_0.InfReleaseUnloading; // from kiln

      A     "MAL1S019Par".Par.FlagFunction_1.StepUnloading; // Step unloading
      AN    "MAL1S019Par".Par.FlagFunction_1.UnloadingStarted;
      A     "G142M".A_2315_BZS22.StFalse; // backwall is not in down pos
      A     "G142M".A_2315_BZS23.StTrue; // backwall is in up pos  // JV030908
      A     "G147M".A_2311_KCL01I5.StTrue; // pushbutton drive fast fwd
      S     "MAL1S019Par".Par.FlagFunction_1.UnloadingStarted;
      FP    "MAL1S019Par".Par.FlagFunction_0.FlagUnloadingStartedFP; // JV030908
      =     "MAL1S019Par".Par.FlagFunction_0.ImpulseUnloadingStarted; // JV030908

      AN    "MAL1S019Par".Par.FlagFunction_1.UnloadingStarted;
      O     "MAL1S019Par".Par.FlagFunction_1.StepCleaning; // Step cleaning
      O     "MAL1S019Par".Par.FlagFunction_1.FinishCleaning;
      JC    EN38;
//BRT250310      L     3600
      L     4000; //BRT250310 -> +2° Overlapping damit die Maschine sicher auf den Endschalter fährt!
      T     "G145M".A_2311_MXZ41MA.Ma.InPositionTarget; // target position unloading
      L     "MAL1S019Par".RecipeHeader.Unloading.UnLoadingSpeed_2; // JV 290808
      T     "MAL1S019Par".Par.ParIntProcess.CopyLoadindSpeed2; // JV 290808
EN38: NOP   0;


NETWORK
TITLE =ASW_8010:  Step unloading finished

// Verweilzeit auf dem Endschalter  =A_2111_BZS44.StTrue --> stop discharge side
//      L     S5T#3M                      // Verweilzeit auf dem Endschalter
//BRT070310      U     "G145M".A_2311_BZS44.StTrue // stop discharge side
      A     "G145M".A_2311_BZS46.StTrue; // stop endposition unloading
//BRT070310      U     "G144M".A_2315_BZS42.StTrue
      A     "G146M".A_2315_MXZ11MA.Ma.StStartedFwd;
//      SE    T    119
//====>BRT070410 - ohne Timer, um Restart der Wartezeit bei Unterbruch Transport zu verhindern!
      AN    "MAL1S019Par".Par.FlagFunction_0.Inf29; //Wartezeit 120s abgelaufen = 1
      A     "SYS_Scan0_Tick1s";
      JCN   wait;
      L     "MAL1S019Par".Par.ParIntMachine.Value33; //aktuelle Wartezeit Maschine bei 100% Unloading-Position
      L     1;
      +I    ;
      T     "MAL1S019Par".Par.ParIntMachine.Value33; //aktuelle Wartezeit Maschine bei 100% Unloading-Position
wait: NOP   0;
      L     "MAL1S019Par".Par.ParIntMachine.Value33; //aktuelle Wartezeit Maschine bei 100% Unloading-Position
      L     120; // 120s
      >=I   ;
      =     "MAL1S019Par".Par.FlagFunction_0.Inf29; //Wartezeit 120s abgelaufen = 1
//<====BRT070410
//************************************************************************************************

      A     "MAL1S019".ToASW.InfDataReady;
      A     "MAL1S019".PCRead.Step.StEmptying;
//====>BRT070310
      A(    ;
      O     "MAL1S019".ToASW.InfSameJobNextSec;
      O(    ;
      L     831; // Next Section: MAL1S031
      L     "MAL1S019".SecNom.HEADER.Kilning_vessel_1; // Target in recipe
      ==I   ;
      )     ;
      )     ;
//<====BRT070310
      A     "MAL1S019Par".Par.FlagFunction_1.StepUnloading; // Step unloading
      AN    "MAL1S019Par".Par.FlagFunction_1.FinishUnloading;
      A     "MAL1S019Par".Par.FlagFunction_1.StepUnloading; // Step unloading
      A     "MAL1S019Par".Par.FlagFunction_1.UnloadingStarted;
//      U     T    119                    // Verweilzeit auf dem Endschalter ist abgelaufen
      A(    ;
      A     "MAL1S019Par".Par.FlagFunction_0.Inf29; //Wartezeit 120s abgelaufen = 1
      O     "MAL1S019".PCWrite.ExtFuncOn.FinishCleanSurface; // PIC command "Finish Unloading"
      )     ;
//------------ Confirmation is necessary to finish unloading **********************
      A(    ;
      L     "G145M".A_2311_MXZ41MA.Ma.OutPositionRel;
      L     950; //95%
      >I    ;
      )     ;
//      U     "MAL1S019".PCWrite.ExtFuncOn.FinishCleanSurface    // PIC command "Finish Unloading"
//************************************************************************************************
      R     "MAL1S019Par".Par.FlagFunction_1.StepUnloading; // Step unloading
      S     "MAL1S019Par".Par.FlagFunction_1.FinishUnloading;
      S     "MAL1S019Par".Par.FlagMachine_0.CmdTurnRevAfterUnloading;
      S     "MAL1S019Par".Par.FlagGen.Flag0024; // finished first unloading
      AN    "MAL1S019Par".Par.FlagMachine_0.CmdTurnRevAfterUnloading;
      JC    EN39;
      L     3399; // 3399 = 94,5%
      T     "G145M".A_2311_MXZ41MA.Ma.InPositionTarget; // target position
EN39: NOP   0;

NETWORK
TITLE =ASW_9000: Step cleaning germination box

      A     "MAL1S019".ToASW.InfDataReady;
      A(    ;
      A     "MAL1S019".PCRead.Step.StEmptied;
      O     "MAL1S019".PCRead.Step.StEmptying;
      )     ;
      A     "MAL1S019Par".Par.FlagFunction_1.FinishUnloading;
      A     "MAL1S019Par".Par.FlagMachine_0.CmdTurnRevAfterUnloading;
      AN    "MAL1S019Par".Par.FlagMachine_0.CleaningAfterUnloading;
      A(    ;
      L     "G145M".A_2311_MXZ41MA.Ma.OutPositionRel;
      L     965; // 956 alt UK 05.11.2010
      <=I   ; // cleaning pos
      )     ;
      A     "G145M".A_2311_BZS46.StFalse; // stop endposition unloading //JV040310
      A     "MAL1S019Par".Par.FlagGen.Flag0024; // finished first unloading
      AN    "MAL1S019Par".Par.FlagGen.Flag0025; // wait pos. to unloading leftover
      AN    "MAL1S019Par".Par.FlagGen.Flag0026; // unloading leftover
      AN    "MAL1S019Par".Par.FlagGen.Flag0027; // finished unloading leftover
      O     "MAL1S019".PCWrite.ExtFuncOn.FinishCleanSurface; // PIC command "Finish Unloading"
      R     "MAL1S019Par".Par.FlagMachine_0.CmdTurnRevAfterUnloading;
      R     "MAL1S019Par".Par.FlagGen.Flag0024; // finished first unloading
      S     "MAL1S019Par".Par.FlagGen.Flag0025; // wait pos. to unloading leftover

//--- Zwischenschritt für Starten einer Restentladung ---
      A     "G147M".A_2311_KCL01I5.StTrue; // pushbutton drive fast fwd
      AN    "MAL1S019Par".Par.FlagGen.Flag0024; // finished first unloading
      A     "MAL1S019Par".Par.FlagGen.Flag0025; // wait pos. to unloading leftover
      AN    "MAL1S019Par".Par.FlagGen.Flag0026; // unloading leftover
      A(    ;
      A     "MAL1S019".PCRead.Step.StEmptied;
      O     "MAL1S019".PCRead.Step.StEmptying;
      )     ;
      A     "MAL1S019Par".Par.FlagFunction_1.FinishUnloading;
      AN    "MAL1S019Par".Par.FlagMachine_0.CmdTurnRevAfterUnloading;
      AN    "MAL1S019Par".Par.FlagMachine_0.CleaningAfterUnloading;
      A(    ;
      L     "G145M".A_2311_MXZ41MA.Ma.OutPositionRel;
      L     965; // 956 alt UK 05.11.2010
      <=I   ; // cleaning pos
      )     ;
      A     "G145M".A_2311_BZS46.StFalse; // stop endposition unloading
      O     "MAL1S019".PCWrite.ExtFuncOn.FinishCleanSurface; // PIC command "Finish Unloading"
      R     "MAL1S019Par".Par.FlagMachine_0.CmdTurnRevAfterUnloading;
      R     "MAL1S019Par".Par.FlagGen.Flag0025; // wait pos. to unloading leftover
      S     "MAL1S019Par".Par.FlagGen.Flag0026; // unloading leftover

      AN    "MAL1S019Par".Par.FlagGen.Flag0026; // unloading leftover
      JC    EN40;
      L     4000;
      T     "G145M".A_2311_MXZ41MA.Ma.InPositionTarget; // target position
EN40: NOP   0;

//--- Erreichen der Endposition nach Restentladung ---
      A     "G145M".A_2311_BZS46.StTrue; // stop endposition unloading
      A     "MAL1S019Par".Par.FlagFunction_1.FinishUnloading;
      A     "MAL1S019Par".Par.FlagGen.Flag0026; // unloading leftover
      A(    ;
      L     "G145M".A_2311_MXZ41MA.Ma.OutPositionRel;
      L     950; //95%
      >I    ;
      )     ;
      O     "MAL1S019".PCWrite.ExtFuncOn.FinishCleanSurface; // PIC command "Finish Unloading"
      R     "MAL1S019Par".Par.FlagGen.Flag0026; // unloading leftover
      S     "MAL1S019Par".Par.FlagGen.Flag0027; // finished unloading leftover
      S     "MAL1S019Par".Par.FlagMachine_0.CmdTurnRevAfterUnloading;

//********************************************************************************************

      A     "MAL1S019".ToASW.InfDataReady;
//====>BRT040310
      A(    ;
      A     "MAL1S019".PCRead.Step.StEmptied;
      O     "MAL1S019".PCRead.Step.StEmptying;
      )     ;
//<====BRT040310
      A     "MAL1S019Par".Par.FlagFunction_1.FinishUnloading;
      A     "MAL1S019Par".Par.FlagMachine_0.CmdTurnRevAfterUnloading;
      AN    "MAL1S019Par".Par.FlagMachine_0.CleaningAfterUnloading;
      A(    ;
      L     "G145M".A_2311_MXZ41MA.Ma.OutPositionRel;
      L     965; // 956 alt UK 05.11.2010
      <=I   ; // cleaning pos
      )     ;
      A     "G145M".A_2311_BZS46.StFalse; // stop endposition unloading //JV040310
//====>BRT120510
      AN    "MAL1S019Par".Par.FlagGen.Flag0024; // finished first unloading
      AN    "MAL1S019Par".Par.FlagGen.Flag0025; // wait pos. to unloading leftover
      AN    "MAL1S019Par".Par.FlagGen.Flag0026; // unloading leftover
      A     "MAL1S019Par".Par.FlagGen.Flag0027; // finished unloading leftover
      O     "MAL1S019".PCWrite.ExtFuncOn.FinishCleanSurface; // PIC command "Finish Unloading"
      R     "MAL1S019Par".Par.FlagGen.Flag0027; // finished unloading leftover
//<====BRT120510
      R     "MAL1S019Par".Par.FlagMachine_0.CmdTurnRevAfterUnloading;
      R     "MAL1S019Par".Par.FlagFunction_1.FinishUnloading;
      S     "MAL1S019Par".Par.FlagMachine_0.CleaningAfterUnloading;
      S     "MAL1S019Par".Par.FlagFunction_1.StepCleaning; // Step cleaning

      SET   ;
      R     "MAL1S019".PCWrite.ExtFuncOn.FinishCleanSurface; // PIC command "Finish Unloading"

NETWORK
TITLE =ASW_9010: Cleaning Germination box finished
//
      A     "MAL1S019".ToASW.InfDataReady;
//====>BRT070310
      A(    ;
      A     "MAL1S019".PCRead.Step.StEmptied;
      O     "MAL1S019".PCRead.Step.StEmptying;
      )     ;
//<====BRT070310
      A     "MAL1S019Par".Par.FlagFunction_1.StepCleaning; // Step cleaning
      A     "G145M".A_2311_BZS44.StFalse; // stop discharge side
      A(    ;
      O     "MAL1S019".PCWrite.ExtFuncOn.FinishCleaning; // PIC command "cleaning finished"
// BRT110310      O     "G147M".A_2311_KCL01I4.InpTrue    // pushbutton "drive rev"
      O     "G147M".A_2311_KCL01I6.InpTrue; // pushbutton "drive rev fast"
      )     ;
      R     "MAL1S019Par".Par.FlagMachine_0.CleaningAfterUnloading;
      R     "MAL1S019Par".Par.FlagFunction_1.StepCleaning; // Step cleaning
      S     "MAL1S019Par".Par.FlagFunction_1.FinishCleaning;

      SET   ;
      R     "MAL1S019".PCWrite.ExtFuncOn.FinishCleaning; // PIC command "cleaning finished"

      A     "MAL1S019".PCRead.Step.StIdling;
//BRT070310      U     "G145M".A_2311_BZS46.StTrue // stop fan side (home pos)
      A     "G145M".A_2311_BZS44.StTrue; // stop zeroposition (home pos)
      A(    ; //dyk 081031 50 pulses
      L     "G145M".A_2311_MXZ41MA.IncCounter.InpActCount;
      L     50;
      <I    ;
      )     ;
      R     "MAL1S019Par".Par.FlagFunction_1.FinishCleaning;

      AN    "MAL1S019Par".Par.FlagFunction_1.FinishCleaning;
      JC    EN41;
      L     0;
      T     "G145M".A_2311_MXZ41MA.Ma.InPositionTarget; // target position
//MW 2008.10.24
      L     "MAL1S019Par".RecipeHeader.Unloading.UnLoadingSpeed_2;
      T     "MAL1S019Par".Par.ParIntProcess.CopyLoadindSpeed2;
EN41: NOP   0;

NETWORK
TITLE =ASW_9080: Send section date to PIC after germination

      OPN   "MAL1S019";
      A     "MAL1S019".PCRead.Step.StEmptying;
      FP    "MAL1S019Par".Par.FlagProcess.FP_SendResultToPIC;
      JCN   E908;
//

E908: NOP   0;
NETWORK
TITLE =ASW_10000: ILO functions

      A     "MAL1S019".SecAc.Sta1On.Inf08;
      =     "MAL1S019".Gr.All.Spare04;

// reset ILO with start unloading   JV080908    special on SALADIN BOXES
      A     "MAL1S019Par".Par.FlagFunction_0.ImpulseUnloadingStarted; // JV030908
      R     "MAL1S019".SecAc.Sta1On.Inf08;

//- Little help for PIC-People
      A     "MAL1S019".SecAc.Sta1On.Inf08;
      JC    RSM;
      L     0;
      T     "MAL1S019Par".Ilo.Code_ILO_Funktion0; // FCM 19 LINE 1 SEC 19 GERM 3
RSM:  NOP   0;
//- Combination OLD and NEW ---
      A     "MAL1S019".SecAc.Sta1On.Inf08;
      JCN   IFM;
      L     "MAL1S019Par".Ilo.ILOMode;
      L     100;
      *I    ;
      T     "MAL1S019Par".Ilo.Code_ILO_Funktion0;
IFM:  NOP   0;

//  no ILO-mode >> cmd manual off to all used groups and reset all flags
      A     "MAL1S019".SecAc.Sta1On.Inf08;
      FN    "MAL1S019Par".Ilo.Flag.EdgeILOModeOn; //BRT070310
//BRT070310      FN    DB907.DBX 3692.0
//      S     DB909.DBX 3006.0            // (ManOff)
//      R     DB909.DBX 3014.0
//      R     DB909.DBX 3018.1
//  Gr-cmd manual OFF
      S     "G007G".Gr.CmdManualOff; // GENERAL ELEMENTS GERM 3
      S     "G142M".Gr.CmdManualOff; // LIFTING DEVICE GERM 3
      S     "G143M".Gr.CmdManualOff; // COUPLING DEVICE TURNER GERM 3
      S     "G144M".Gr.CmdManualOff; // COUPLING DEVICE WALL GERM 3
      S     "G145M".Gr.CmdManualOff; // TRAVELLING DRIVE GERM 3
      S     "G146M".Gr.CmdManualOff; // HORIZONTAL AND LIFTING SCREW GERM 3
      S     "G149M".Gr.CmdManualOff; // TURNING SCREWS GERM 3
      S     "G150M".Gr.CmdManualOff; // FAN AND VALVE SRAY AIR GERM 3
//      S     "G151M".Gr.CmdManualOff     // FRESH AIR LOUVER GERM 3
      S     "G152M".Gr.CmdManualOff; // EXHAUST AIR LOUVER GERM 3
      S     "G157M".Gr.CmdManualOff; // COOLING / HEATING GERM 3
//  RESET ADDITIONAL CMD`S
      R     "G142M".USW14; // ILO-cmd
      R     "G142M".USW15; // ILO-cmd
      R     "G143M".USW14; // ILO-cmd
      R     "G143M".USW15; // ILO-cmd
      R     "G144M".USW14; // ILO-cmd
      R     "G144M".USW15; // ILO-cmd
      R     "G145M".USW14; // ILO-cmd
      R     "G145M".USW15; // ILO-cmd
      R     "G146M".USW14; // ILO-cmd
      R     "G146M".USW15; // ILO-cmd
      R     "G149M".USW14; // ILO-cmd
      R     "G149M".USW15; // ILO-cmd
      R     "G150M".USW14; // ILO-cmd
      R     "G150M".USW15; // ILO-cmd
      R     "G151M".USW14; // ILO-cmd
      R     "G151M".USW15; // ILO-cmd
      R     "G152M".USW14; // ILO-cmd
      R     "G152M".USW15; // ILO-cmd
      R     "G157M".USW14; // ILO-cmd
      R     "G157M".USW15; // ILO-cmd

      A     "MAL1S019".SecAc.Sta1On.Inf08;
      JC    RSM2;
      L     0;
      T     #tmpInt;
      CALL "SIEMENS_FILL" (
           BVAL                     := #tmpInt,
           RET_VAL                  := #tmpRET,
           BLK                      := "MAL1S019Par".Ilo);
RSM2: NOP   0;


      NOP   0;
// --- FCM 04 - Fans ---
      L     "MAL1S019Par".Ilo.ILOMode;
      L     4;
      <>I   ;
      JC    IO4;
// man on
      A     "MAL1S019Par".Ilo.GrCMDManOn[1];
      S     "G150M".Gr.InManual; // FAN AND VALVE SRAY AIR GERM 3
      S     "G151M".Gr.InManual; // FRESH AIR LOUVER GERM 3
      S     "G152M".Gr.InManual; // EXHAUST AIR LOUVER GERM 3
      R     "MAL1S019Par".Ilo.GrCMDManOn[1];
// man off
      A     "MAL1S019Par".Ilo.GrCMDManOff[1];
      S     "G150M".Gr.CmdManualOff; // FAN AND VALVE SRAY AIR GERM 3
      R     "G150M".Gr.InManual; // FAN AND VALVE SRAY AIR GERM 3
      R     "G150M".USW14; // ILO-cmd
      R     "G150M".USW15; // ILO-cmd
      S     "G151M".Gr.CmdManualOff; // FRESH AIR LOUVER GERM 3
      R     "G151M".Gr.InManual; // FRESH AIR LOUVER GERM 3
      R     "G151M".USW14; // ILO-cmd
      R     "G151M".USW15; // ILO-cmd
      S     "G152M".Gr.CmdManualOff; // EXHAUST AIR LOUVER GERM 3
      R     "G152M".Gr.InManual; // EXHAUST AIR LOUVER GERM 3
      R     "G152M".USW14; // ILO-cmd
      R     "G152M".USW15; // ILO-cmd
      R     "MAL1S019Par".Ilo.GrCMDManOff[1];
      R     "MAL1S019Par".Ilo.GrCMDManAdditional.Cmd1[1];
      R     "MAL1S019Par".Ilo.GrCMDManAdditional.Cmd2[1];
// man start
      A     "MAL1S019Par".Ilo.GrCMDManStart[1];
      S     "G150M".Gr.CmdOn; // FAN AND VALVE SRAY AIR GERM 3
      S     "G150M".Gr.CmdContinue; // FAN AND VALVE SRAY AIR GERM 3
      S     "G151M".Gr.CmdOn; // FRESH AIR LOUVER GERM 3
      S     "G151M".Gr.CmdContinue; // FRESH AIR LOUVER GERM 3
      S     "G152M".Gr.CmdOn; // EXHAUST AIR LOUVER GERM 3
      S     "G152M".Gr.CmdContinue; // EXHAUST AIR LOUVER GERM 3
      R     "MAL1S019Par".Ilo.GrCMDManStart[1];
      A     "MAL1S019Par".Ilo.GrCMDManStart[2];
      R     "MAL1S019Par".Ilo.GrCMDManStart[2];
// man stop
      A     "MAL1S019Par".Ilo.GrCMDManStop[1];
      S     "G150M".Gr.CmdOff; // FAN AND VALVE SRAY AIR GERM 3
//BRT070310      S     "G150M".Gr.CmdOff           // FRESH AIR LOUVER GERM 3
//BRT070310      S     "G150M".Gr.CmdOff           // EXHAUST AIR LOUVER GERM 3
      R     "MAL1S019Par".Ilo.GrCMDManStop[1];
// man fault reset
//BRT070310      U     "MAL1S019Par".Ilo.GrCMDManOn[17]
      A     "MAL1S019Par".Ilo.GrCMDManFaultReset[1]; //BRT070310
      S     "G150M".Gr.CmdFaultReset; // FAN AND VALVE SRAY AIR GERM 3
      S     "G151M".Gr.CmdFaultReset; // FRESH AIR LOUVER GERM 3
      S     "G152M".Gr.CmdFaultReset; // EXHAUST AIR LOUVER GERM 3
      R     "MAL1S019Par".Ilo.GrCMDManFaultReset[1];
// target position
      AN    "G150M".Gr.InManual; // FAN AND VALVE SRAY AIR GERM 3
      O(    ;
      L     "MAL1S019Par".Ilo.Code_ILO_Funktion0;
      L     400;
      <>I   ;
      )     ;
      JC    F04a;
      L     "MAL1S019Par".Ilo.SetpointInt01[1];
      T     "MAL1S019Par".Par.ParIntProcess.Speed_ILO_Fan;
F04a: NOP   0;
//BRT070310 - Sollwert Frischluftklappen!
      AN    "G151M".Gr.InManual; // FRESH AIR LOUVER GERM 3
      O(    ;
      L     "MAL1S019Par".Ilo.Code_ILO_Funktion0;
      L     400;
      <>I   ;
      )     ;
      JC    F04b;
      L     "MAL1S019Par".Ilo.SetpointInt02[1];
      T     "MAL1S019Par".Par.ParIntProcess.TarPos_ILO_FreshAir;
F04b: NOP   0;

IO4:  NOP   0;
      NOP   0;
// --- FCM 05 - Fans with target air temperature ---
      L     "MAL1S019Par".Ilo.ILOMode;
      L     5;
      <>I   ;
      JC    IO5;
// man on
      A     "MAL1S019Par".Ilo.GrCMDManOn[1];
      S     "G150M".Gr.InManual; // FAN AND VALVE SRAY AIR GERM 3
      S     "G151M".Gr.InManual; // FRESH AIR LOUVER GERM 3
      S     "G152M".Gr.InManual; // EXHAUST AIR LOUVER GERM 3  //BRT070310
      S     "G157M".Gr.InManual; // COOLING / HEATING GERM 3
      R     "MAL1S019Par".Ilo.GrCMDManOn[1];
// man off
      A     "MAL1S019Par".Ilo.GrCMDManOff[1];
      S     "G150M".Gr.CmdManualOff; // FAN AND VALVE SRAY AIR GERM 3
      R     "G150M".Gr.InManual; // FAN AND VALVE SRAY AIR GERM 3
      R     "G150M".USW14; // ILO-cmd
      R     "G150M".USW15; // ILO-cmd
      S     "G151M".Gr.CmdManualOff; // FRESH AIR LOUVER GERM 3
      R     "G151M".Gr.InManual; // FRESH AIR LOUVER GERM 3
      R     "G151M".USW14; // ILO-cmd
      R     "G151M".USW15; // ILO-cmd
      S     "G152M".Gr.CmdManualOff; // EXHAUST AIR LOUVER GERM 3  //BRT070310
      R     "G152M".Gr.InManual; // EXHAUST AIR LOUVER GERM 3  //BRT070310
      R     "G152M".USW14; // ILO-cmd                    //BRT070310
      R     "G152M".USW15; // ILO-cmd                    //BRT070310
      S     "G157M".Gr.CmdManualOff; // COOLING / HEATING GERM 3
      R     "G157M".Gr.InManual; // COOLING / HEATING GERM 3
      R     "G157M".USW14; // ILO-cmd
      R     "G157M".USW15; // ILO-cmd
      R     "MAL1S019Par".Ilo.GrCMDManOff[1];
      R     "MAL1S019Par".Ilo.GrCMDManAdditional.Cmd1[1];
      R     "MAL1S019Par".Ilo.GrCMDManAdditional.Cmd2[1];
// man start
      A     "MAL1S019Par".Ilo.GrCMDManStart[1];
      S     "G150M".Gr.CmdOn; // FAN AND VALVE SRAY AIR GERM 3
      S     "G150M".Gr.CmdContinue; // FAN AND VALVE SRAY AIR GERM 3
      S     "G151M".Gr.CmdOn; // FRESH AIR LOUVER GERM 3
      S     "G151M".Gr.CmdContinue; // FRESH AIR LOUVER GERM 3
      S     "G152M".Gr.CmdOn; // EXHAUST AIR LOUVER GERM 3   //BRT070310
      S     "G152M".Gr.CmdContinue; // EXHAUST AIR LOUVER GERM 3   //BRT070310
      S     "G157M".Gr.CmdOn; // COOLING / HEATING GERM 3
      S     "G157M".Gr.CmdContinue; // COOLING / HEATING GERM 3
      R     "MAL1S019Par".Ilo.GrCMDManStart[1];
      A     "MAL1S019Par".Ilo.GrCMDManStart[2];
      R     "MAL1S019Par".Ilo.GrCMDManStart[2];
// man stop
      A     "MAL1S019Par".Ilo.GrCMDManStop[1];
      S     "G150M".Gr.CmdOff; // FAN AND VALVE SRAY AIR GERM 3
//BRT070310      S     "G151M".Gr.CmdOff           // FRESH AIR LOUVER GERM 3
//BRT070310      S     "G152M".Gr.CmdOff           // EXHAUST AIR LOUVER GERM 3
      S     "G157M".Gr.CmdOff; // COOLING / HEATING GERM 3
      R     "MAL1S019Par".Ilo.GrCMDManStop[1];
// man fault reset
      A     "MAL1S019Par".Ilo.GrCMDManFaultReset[1];
      S     "G150M".Gr.CmdFaultReset; // FAN AND VALVE SRAY AIR GERM 3
      S     "G151M".Gr.CmdFaultReset; // FRESH AIR LOUVER GERM 3
      S     "G152M".Gr.CmdFaultReset; // EXHAUST AIR LOUVER GERM 3   //BRT070310
      S     "G157M".Gr.CmdFaultReset; // COOLING / HEATING GERM 3
      R     "MAL1S019Par".Ilo.GrCMDManFaultReset[1];
// target position
      AN    "G157M".Gr.InManual; // COOLING / HEATING GERM 3
      JC    F05a;
      L     "MAL1S019Par".Ilo.SetpointInt02[1];
      T     "MAL1S019Par".Par.ParIntProcess.TargetTemperature_ILO;
F05a: NOP   0;
      AN    "G150M".Gr.InManual; // FAN AND VALVE SRAY AIR GERM 3
      O(    ;
      L     "MAL1S019Par".Ilo.Code_ILO_Funktion0;
      L     500;
      <>I   ;
      )     ;
      JC    F05b;
      L     "MAL1S019Par".Ilo.SetpointInt01[1];
      T     "MAL1S019Par".Par.ParIntProcess.Speed_ILO_Fan;
F05b: NOP   0;
//BRT070310 - Sollwert Frischluftklappen!
      AN    "G151M".Gr.InManual; // FRESH AIR LOUVER GERM 3
      O(    ;
      L     "MAL1S019Par".Ilo.Code_ILO_Funktion0;
      L     500;
      <>I   ;
      )     ;
      JC    F05c;
      L     "MAL1S019Par".Ilo.SetpointInt03[1];
      T     "MAL1S019Par".Par.ParIntProcess.TarPos_ILO_FreshAir;
F05c: NOP   0;

IO5:  NOP   0;
      NOP   0;
// --- FCM 06 - Fresh air flap ---
      L     "MAL1S019Par".Ilo.ILOMode;
      L     6;
      <>I   ;
      JC    IO6;
// man on
      A     "MAL1S019Par".Ilo.GrCMDManOn[1];
      S     "G151M".Gr.InManual; // FRESH AIR LOUVER GERM 3
//      R     DB909.DBX 3032.0
// man off
      A     "MAL1S019Par".Ilo.GrCMDManOff[1];
      S     "G151M".Gr.CmdManualOff; // FRESH AIR LOUVER GERM 3
      R     "G151M".Gr.InManual; // FRESH AIR LOUVER GERM 3
      R     "G151M".USW14; // ILO-cmd
      R     "G151M".USW15; // ILO-cmd
      R     "MAL1S019Par".Ilo.GrCMDManOff[1];
      R     "MAL1S019Par".Ilo.GrCMDManAdditional.Cmd1[1];
      R     "MAL1S019Par".Ilo.GrCMDManAdditional.Cmd2[1];
// man start
      A     "MAL1S019Par".Ilo.GrCMDManStart[1];
      S     "G151M".Gr.CmdOn; // FRESH AIR LOUVER GERM 3
      S     "G151M".Gr.CmdContinue; // FRESH AIR LOUVER GERM 3
      R     "MAL1S019Par".Ilo.GrCMDManStart[1];
      A     "MAL1S019Par".Ilo.GrCMDManStart[2];
      R     "MAL1S019Par".Ilo.GrCMDManStart[2];

      A     "MAL1S019Par".Ilo.GrCMDManOn[1];
      R     "MAL1S019Par".Ilo.GrCMDManOn[1];
// man stop
      A     "MAL1S019Par".Ilo.GrCMDManStop[1];
      S     "G151M".Gr.CmdOff; // FRESH AIR LOUVER GERM 3
      R     "MAL1S019Par".Ilo.GrCMDManStop[1];
// man fault reset
//BRT070310      U     "MAL1S019Par".Ilo.GrCMDManOn[17]
      A     "MAL1S019Par".Ilo.GrCMDManFaultReset[1]; //BRT070310
      S     "G151M".Gr.CmdFaultReset; // FRESH AIR LOUVER GERM 3
      R     "MAL1S019Par".Ilo.GrCMDManOn[17];
// moving direction

// target position
      AN    "G151M".Gr.InManual; // FRESH AIR LOUVER GERM 3
      JC    F06b;
      L     "MAL1S019Par".Ilo.SetpointInt01[1];
      T     "MAL1S019Par".Par.ParIntProcess.TarPos_ILO_FreshAir;
F06b: NOP   0;

